(* IEC 61131-3 sources: SmartHomeNew/snapshots/2026-05-05, 45 files *)

(* ---- E_Lifetime_Device_Type.dut ---- *)
{attribute 'strict'}
TYPE E_Lifetime_Device_Type :
(
    LIFETIME_DEVICE_PUMP := 1,
    LIFETIME_DEVICE_FAN  := 2
) USINT;
END_TYPE

(* ---- E_Rule_Action_Type.dut ---- *)
{attribute 'strict'}
TYPE E_Rule_Action_Type :
(
    ACTION_NONE := 0,
    ACTION_SET_FLOOR_HEATING := 1,
    ACTION_SET_LIGHTING_BASE := 2,
    ACTION_SET_LIGHTING_ACCENT := 3,
    ACTION_SET_SOCKET := 4,
    ACTION_SET_VENTILATION := 5,
    ACTION_SET_BLINDS := 6,
    ACTION_ACTIVATE_SCENARIO := 7,
    ACTION_TOGGLE_LIGHTING := 8,
    ACTION_TOGGLE_SOCKET := 9
) USINT;
END_TYPE

(* ---- E_SCENARIO_SOURCE.dut ---- *)
TYPE E_SCENARIO_SOURCE :
(
    SRC_NONE := 0,
    SRC_OPERATOR := 1,
    SRC_GATEWAY := 2,
    SRC_RULE := 3,
    SRC_SAFETY := 4,
    SRC_POLICY := 5
);
END_TYPE

(* ---- E_System_Severity.dut ---- *)
TYPE E_System_Severity :
(
    SEV_NORMAL,
    SEV_WARNING,
    SEV_DEGRADED,
    SEV_CRITICAL
);
END_TYPE

(* ---- E_Trace_Source.dut ---- *)
{attribute 'strict'}
TYPE E_Trace_Source :
(
    SRC_MAIN := 0,
    SRC_IO := 1,
    SRC_DIAGNOSTICS := 2,
    SRC_HEATING := 3,
    SRC_SCENARIO := 4,
    SRC_USER := 5
) USINT;
END_TYPE

(* ---- GVL_SAFETY_SHUTDOWN.gvl ---- *)
TYPE E_Safety_Mode :
(
    NORMAL,
    FIRE,
    GAS,
    WATER_LEAK,
    GLOBAL_STOP,
    EVACUATION
);
END_TYPE

VAR_GLOBAL
    G_Safety_Mode : E_Safety_Mode := NORMAL;
    G_Safety_Active : BOOL := FALSE;
END_VAR

(* ---- GVL_CONFIG_CONTROL.gvl ---- *)
{attribute 'qualified_only'}
VAR_GLOBAL
    // Config change control. HMI/service writes here, never directly to active safety config.

    G_Apply_Request : BOOL := FALSE;
    G_Apply_Confirm : BOOL := FALSE;
    G_Rollback_Request : BOOL := FALSE;
    G_Rollback_Confirm : BOOL := FALSE;
    G_Reset_Default_Request : BOOL := FALSE;
    G_Reset_Default_Confirm : BOOL := FALSE;

    G_Config_Version : UDINT := 1;
    G_Last_Good_Version : UDINT := 1;
    G_Backup_Valid : BOOL := FALSE;
    G_Apply_Done : BOOL := FALSE;
    G_Rollback_Done : BOOL := FALSE;

    // STAGED INPUT CONFIG
    STG_Reputation_Learning_Rate : REAL := 0.05;
    STG_Reputation_Recovery_Decay : REAL := 0.01;
    STG_Min_Sensor_Confidence : REAL := 0.1;
    STG_Bad_Spike_Confidence : REAL := 0.3;
    STG_Default_Confidence : REAL := 1.0;

    // STAGED SCENARIO CONFIG
    STG_Night_Start_Hour : INT := 22;
    STG_Night_End_Hour : INT := 6;
    STG_VentBoost_Humidity_Threshold : REAL := 65.0;

    // STAGED RECOVERY CONFIG
    STG_Stabilization_Delay_MS : UDINT := 5000;

    // STAGED COMMAND POLICY CRITICAL PART
    STG_PLC_Inactive_Close_Gas : BOOL := TRUE;
    STG_PLC_Inactive_Stop_Boiler : BOOL := TRUE;
    STG_PLC_Inactive_Block_Heating : BOOL := TRUE;
    STG_PLC_Inactive_Stop_Vent : BOOL := TRUE;
    STG_PLC_Inactive_Block_Water : BOOL := TRUE;

    // BACKUP INPUT CONFIG
    BCK_Reputation_Learning_Rate : REAL := 0.05;
    BCK_Reputation_Recovery_Decay : REAL := 0.01;
    BCK_Min_Sensor_Confidence : REAL := 0.1;
    BCK_Bad_Spike_Confidence : REAL := 0.3;
    BCK_Default_Confidence : REAL := 1.0;

    // BACKUP SCENARIO CONFIG
    BCK_Night_Start_Hour : INT := 22;
    BCK_Night_End_Hour : INT := 6;
    BCK_VentBoost_Humidity_Threshold : REAL := 65.0;

    // BACKUP RECOVERY CONFIG
    BCK_Stabilization_Delay_MS : UDINT := 5000;

    // BACKUP COMMAND POLICY CRITICAL PART
    BCK_PLC_Inactive_Close_Gas : BOOL := TRUE;
    BCK_PLC_Inactive_Stop_Boiler : BOOL := TRUE;
    BCK_PLC_Inactive_Block_Heating : BOOL := TRUE;
    BCK_PLC_Inactive_Stop_Vent : BOOL := TRUE;
    BCK_PLC_Inactive_Block_Water : BOOL := TRUE;
END_VAR

(* ---- GVL_HEATING_OUTPUT.gvl ---- *)
VAR_GLOBAL
    // Heating output projection produced by PRG_Heating and consumed by PRG_IO_Write.
    // This removes the direct PRG_IO_Write -> GVL_STATE dependency for Heating physical outputs.

    DO_Zone_Valves : ARRAY[1..GVL_CONSTANTS.C_MAX_HEATING_CIRCUITS] OF BOOL;
    DO_Manifold_Pumps : ARRAY[1..GVL_CONSTANTS.C_MAX_MANIFOLDS] OF BOOL;
    AO_Manifold_Valves : ARRAY[1..GVL_CONSTANTS.C_MAX_MANIFOLDS] OF UINT;

    DO_DHW_Heating_Pump : BOOL := FALSE;
    DO_DHW_Circ_Pump : BOOL := FALSE;
    DO_Backup_Circulation_Pump : BOOL := FALSE;
    DO_Electric_Heater_Enable : BOOL := FALSE;
END_VAR

(* ---- GVL_HMI.gvl ---- *)
{attribute 'qualified_only'}
VAR_GLOBAL
    // Heating dashboard
    G_HMI_Heating_Confidence : REAL := 1.0;
    G_HMI_Heating_Confidence_Percent : INT := 100;
    G_HMI_Heating_Reason_Code : INT := 0;
    G_HMI_Heating_Status_Text : STRING(128) := 'OK';
    G_HMI_Heating_Status_Level : INT := 0; // 0=OK, 1=WARN, 2=ALARM

    // Heating predictive dashboard
    G_HMI_Heating_Predictive_Pressure_Drop : ARRAY[1..GVL_CONSTANTS.C_MAX_MANIFOLDS] OF BOOL;
    G_HMI_Heating_Predictive_Current_Rise : ARRAY[1..GVL_CONSTANTS.C_MAX_MANIFOLDS] OF BOOL;
END_VAR

(* ---- GVL_INTENT_BEHAVIOR.gvl ---- *)
VAR_GLOBAL
    // Behavior / Scenario Engine intent layer.
    // Scenario Engine writes here; Command Arbitration may consume it.

    I_Request_Night_Mode : BOOL := FALSE;
    I_Request_Away_Mode : BOOL := FALSE;
    I_Request_Comfort_Mode : BOOL := FALSE;
    I_Request_Energy_Save_Mode : BOOL := FALSE;
    I_Request_Preheat : BOOL := FALSE;
    I_Request_Ventilation_Boost : BOOL := FALSE;
    I_Request_Access_Secure_Mode : BOOL := FALSE;

    I_Target_Comfort_Temperature : REAL := 21.0;
    I_Behavior_Priority : INT := 0;

    // Candidate scenario scores for explainability / diagnostics
    I_Score_Comfort : INT := 0;
    I_Score_Night : INT := 0;
    I_Score_Energy_Save : INT := 0;
    I_Score_Preheat : INT := 0;
    I_Score_Vent_Boost : INT := 0;
    I_Score_Access_Secure : INT := 0;

    // Multi-objective weights, normalized 0.0..1.0 for HMI / downstream blending.
    I_Weight_Comfort : REAL := 0.0;
    I_Weight_Night : REAL := 0.0;
    I_Weight_Energy_Save : REAL := 0.0;
    I_Weight_Preheat : REAL := 0.0;
    I_Weight_Vent_Boost : REAL := 0.0;
    I_Weight_Access_Secure : REAL := 0.0;

    I_Best_VentBoost_Zone : INT := 0;

    I_Selected_Scenario_Code : E_System_Reason_Code := REASON_NONE;
    I_Selected_Scenario_Text : STRING(255) := 'No behavior scenario selected';

    I_Reason_Code : E_System_Reason_Code := REASON_NONE;
    I_Reason_Text : STRING(255) := 'No behavior scenario active';
    I_Last_Update_MS : UDINT := 0;
END_VAR

(* ---- GVL_INTENT_SAFETY.gvl ---- *)
VAR_GLOBAL
    // --- meta / traceability ---
    I_Source_Valid : BOOL := FALSE;
    I_Last_Update_Cycle : UDINT := 0;
    I_Last_Update_MS : UDINT := 0;

    // --- safety facts for arbitration ---
    I_Fire_Alarm_Active : BOOL := FALSE;
    I_Gas_Alarm_Active : BOOL := FALSE;
    I_Leak_Alarm_Active : BOOL := FALSE;
    I_CO_Warning_Active : BOOL := FALSE;
    I_System_Safe_Stop_Required : BOOL := FALSE;
    I_Freeze_Protection_Required : BOOL := FALSE;
    I_Evacuation_Mode_Active : BOOL := FALSE;

    // --- gas / boiler / ventilation constraints ---
    I_Gas_Close_Required : BOOL := FALSE;
    I_Boiler_Stop_Required : BOOL := FALSE;
    I_Vent_Stop_Required : BOOL := FALSE;
    I_Vent_Force_PV3_Boost : BOOL := FALSE;
    I_Vent_Force_Supply_100 : BOOL := FALSE;
    I_Vent_Force_Supply_80 : BOOL := FALSE;
    I_Vent_Force_Exhaust_100 : BOOL := FALSE;

    // --- water constraints ---
    I_Water_Main_Close_Required : BOOL := FALSE;
    I_Water_Zone_Close_Required : ARRAY[1..32] OF BOOL;
    I_Water_Selective_Recovery_Allowed : BOOL := FALSE;
    I_Water_Recovery_Target_Zone : INT := 0;

    // --- lock / evacuation constraints ---
    I_Lock_1_Force_Open : BOOL := FALSE;
    I_Lock_1_Force_Close_Block : BOOL := FALSE;
    I_Lock_2_Force_Open : BOOL := FALSE;
    I_Lock_2_Force_Close_Block : BOOL := FALSE;
    // --- operator / test constraints ---
    I_Test_Timeout_Gas_Close : BOOL := FALSE;
    I_Test_Timeout_Water_Close : BOOL := FALSE;
END_VAR

(* ---- GVL_SIMULATION.gvl ---- *)
{attribute 'qualified_only'}
VAR_GLOBAL
    G_Simulation_Enable : BOOL := FALSE;

    // Scenario control
    G_Test_Scenario_ID : INT := 0; // 0=manual flags, 1=safety gas, 2=leak+low pressure, 3=sensor+predictive, 4=dual PLC, 5=full stress
    G_Test_Start : BOOL := FALSE;
    G_Test_Stop : BOOL := FALSE;
    G_Test_Scenario_Active : BOOL := FALSE;
    G_Test_Started_MS : UDINT := 0;
    G_Test_Duration_MS : UDINT := 30000;
    G_Test_Expected_Result_Code : INT := 0; // 0=none, 1=safety, 2=heating degraded, 3=role conflict, 4=full stress

    // Sensor fault injection requests
    G_Inject_Heating_Sensor_Fault : BOOL := FALSE;
    G_Inject_IO_Fault : BOOL := FALSE;
    G_Inject_Low_Pressure : BOOL := FALSE;
    G_Inject_Predictive_Pump_Fault : BOOL := FALSE;

    // Safety fault injection requests
    G_Inject_Gas_Alarm : BOOL := FALSE;
    G_Inject_Leak_Alarm : BOOL := FALSE;
    G_Inject_Smoke_Alarm : BOOL := FALSE;

    // PLC / role fault injection request
    G_Inject_Dual_PLC_Active : BOOL := FALSE;

    // Isolated effective simulation outputs. Production state is not overwritten by PRG_System_Simulation.
    G_Sim_Heating_Sensor_Fault : BOOL := FALSE;
    G_Sim_IO_Fault : BOOL := FALSE;
    G_Sim_Low_Pressure : BOOL := FALSE;
    G_Sim_Predictive_Pump_Fault : BOOL := FALSE;
    G_Sim_Gas_Alarm : BOOL := FALSE;
    G_Sim_Leak_Alarm : BOOL := FALSE;
    G_Sim_Smoke_Alarm : BOOL := FALSE;
    G_Sim_Dual_PLC_Active : BOOL := FALSE;

    // Test status
    G_Test_Running : BOOL := FALSE;
    G_Test_Result_OK : BOOL := FALSE;
    G_Test_Last_Result_Text : STRING(128) := 'No test executed';
END_VAR

(* ---- GVL_SYSTEM_SIZE_CONFIG.gvl ---- *)
{attribute 'qualified_only'}
VAR_GLOBAL
    // Runtime active counts. Arrays remain allocated by GVL_CONSTANTS.C_MAX_*.
    // These values define how many channels/zones are actively processed.

    G_Active_Heating_Circuits : INT := GVL_CONSTANTS.C_MAX_HEATING_CIRCUITS;
    G_Active_Water_Zones : INT := GVL_CONSTANTS.C_MAX_WATER_ZONES;
    G_Active_Light_Zones : INT := GVL_CONSTANTS.C_MAX_LIGHT_ZONES;
    G_Active_Blinds : INT := GVL_CONSTANTS.C_MAX_BLINDS;
    G_Active_Sockets : INT := GVL_CONSTANTS.C_MAX_SOCKETS;
END_VAR

(* ---- FB_Boiler_OpenTherm_Interface.st ---- *)
FUNCTION_BLOCK FB_Boiler_OpenTherm_Interface
VAR_INPUT
    VI_Enable : ARRAY[1..GVL_CONSTANTS.C_MAX_BOILERS] OF BOOL;
    VI_Setpoint : ARRAY[1..GVL_CONSTANTS.C_MAX_BOILERS] OF REAL;

    VI_OT_Online : ARRAY[1..GVL_CONSTANTS.C_MAX_BOILERS] OF BOOL;
    VI_OT_Error : ARRAY[1..GVL_CONSTANTS.C_MAX_BOILERS] OF BOOL;
END_VAR

VAR_OUTPUT
    VO_OT_Enable : ARRAY[1..GVL_CONSTANTS.C_MAX_BOILERS] OF BOOL;
    VO_OT_Setpoint : ARRAY[1..GVL_CONSTANTS.C_MAX_BOILERS] OF REAL;
    VO_OT_Command_Valid : ARRAY[1..GVL_CONSTANTS.C_MAX_BOILERS] OF BOOL;
END_VAR

VAR
    L_i : INT;
END_VAR

FOR L_i := 1 TO GVL_CONSTANTS.C_MAX_BOILERS DO
    VO_OT_Enable[L_i] := FALSE;
    VO_OT_Setpoint[L_i] := 0.0;
    VO_OT_Command_Valid[L_i] := FALSE;

    IF VI_Enable[L_i] AND VI_OT_Online[L_i] AND NOT VI_OT_Error[L_i] THEN
        VO_OT_Enable[L_i] := TRUE;
        VO_OT_Setpoint[L_i] := LIMIT(20.0, VI_Setpoint[L_i], 80.0);
        VO_OT_Command_Valid[L_i] := TRUE;
    END_IF;
END_FOR;
END_FUNCTION_BLOCK

(* ---- FB_Calibration_Manager.st ---- *)
FUNCTION_BLOCK FB_Calibration_Manager
VAR_INPUT
    VI_Raw_Value : REAL;
    VI_Type : BYTE; // 1-Temp, 2-Pressure, 3-Gas
    VI_Calib_Record : ST_Sensor_Calibration_Record;
    VI_System_Time_MS : UDINT;
    VI_Start_Verification : BOOL;
END_VAR
VAR_OUTPUT
    VO_Calibrated_Value : REAL;
    VO_Verification_Active : BOOL;
    VO_Verification_Failed : BOOL;
    VO_Deviation_Percent : REAL;
END_VAR
VAR
    L_Verification_Timer : FB_System_Timer;
    L_Initial_Value : REAL;
END_VAR

// 1. Расчет калиброванного значения
CASE VI_Type OF
    1: VO_Calibrated_Value := VI_Raw_Value + VI_Calib_Record.offset;
    2, 3: VO_Calibrated_Value := (VI_Raw_Value * VI_Calib_Record.multiplier) + VI_Calib_Record.offset;
END_CASE;

// 2. Верификация через 1 час (ТЗ 9.5)
IF VI_Start_Verification AND NOT VO_Verification_Active THEN
    VO_Verification_Active := TRUE;
    L_Initial_Value := VO_Calibrated_Value;
END_IF;

L_Verification_Timer(IN := VO_Verification_Active, PT := T#1h, VI_System_Time_MS := VI_System_Time_MS);

IF L_Verification_Timer.Q THEN
    VO_Verification_Active := FALSE;

    // ТЗ 9.5: Отклонение ≤2.0% (норма) / >5.0% (ошибка)
    IF L_Initial_Value <> 0 THEN
        VO_Deviation_Percent := ABS(VO_Calibrated_Value - L_Initial_Value) / L_Initial_Value * 100.0;
    ELSE
        VO_Deviation_Percent := 0.0;
    END_IF;

    VO_Verification_Failed := (VO_Deviation_Percent > 5.0);
END_IF;
END_FUNCTION_BLOCK

(* ---- FB_Fault_Logger.st ---- *)
FUNCTION_BLOCK FB_Fault_Logger
VAR_INPUT
    VI_Severity  : E_System_Severity;
    VI_RootCause : E_System_Root_Cause;
    VI_Time_MS   : UDINT;
END_VAR

VAR_OUTPUT
    VO_Last_Event_Text : STRING(200);
    VO_Event_Count     : UINT;
    VO_Last_Index      : UINT;

    VO_Event_Time_MS   : ARRAY[1..16] OF UDINT;
    VO_Event_Severity  : ARRAY[1..16] OF E_System_Severity;
    VO_Event_RootCause : ARRAY[1..16] OF E_System_Root_Cause;
    VO_Event_Text      : ARRAY[1..16] OF STRING(200);
END_VAR

VAR
    L_Last_Severity  : E_System_Severity;
    L_Last_RootCause : E_System_Root_Cause;
    L_Write_Index    : UINT := 0;
    L_Event_Text     : STRING(200);
END_VAR

L_Event_Text := '';

IF (VI_Severity <> L_Last_Severity) OR (VI_RootCause <> L_Last_RootCause) THEN
    CASE VI_RootCause OF
        E_System_Root_Cause.ROOT_FIRE:
            L_Event_Text := 'EVENT: FIRE DETECTED';
        E_System_Root_Cause.ROOT_GAS_LEAK:
            L_Event_Text := 'EVENT: GAS LEAK';
        E_System_Root_Cause.ROOT_CO_CRITICAL:
            L_Event_Text := 'EVENT: CO CRITICAL';
        E_System_Root_Cause.ROOT_CO_WARNING:
            L_Event_Text := 'EVENT: CO WARNING';
        E_System_Root_Cause.ROOT_WATER_LEAK:
            L_Event_Text := 'EVENT: WATER LEAK';
        E_System_Root_Cause.ROOT_SENSOR_FAULT:
            L_Event_Text := 'EVENT: SENSOR FAULT';
        E_System_Root_Cause.ROOT_IO_OFFLINE:
            L_Event_Text := 'EVENT: IO OFFLINE';
        E_System_Root_Cause.ROOT_COMM_FAULT:
            L_Event_Text := 'EVENT: COMM FAULT';
        E_System_Root_Cause.ROOT_WATCHDOG_FAULT:
            L_Event_Text := 'EVENT: WATCHDOG FAULT';
        E_System_Root_Cause.ROOT_SUBSYSTEM_FAULT:
            L_Event_Text := 'EVENT: SUBSYSTEM FAULT';
        ELSE
            L_Event_Text := 'EVENT: SYSTEM STATE CHANGE';
    END_CASE;

    L_Write_Index := L_Write_Index + 1;
    IF L_Write_Index > 16 THEN
        L_Write_Index := 1;
    END_IF;

    VO_Event_Time_MS[L_Write_Index] := VI_Time_MS;
    VO_Event_Severity[L_Write_Index] := VI_Severity;
    VO_Event_RootCause[L_Write_Index] := VI_RootCause;
    VO_Event_Text[L_Write_Index] := L_Event_Text;

    VO_Last_Index := L_Write_Index;
    VO_Last_Event_Text := L_Event_Text;

    IF VO_Event_Count < 16 THEN
        VO_Event_Count := VO_Event_Count + 1;
    END_IF;
END_IF;

L_Last_Severity := VI_Severity;
L_Last_RootCause := VI_RootCause;
// >>> BULK_SYNC_ANCHOR: FB_Fault_Logger <<<
END_FUNCTION_BLOCK

(* ---- FB_FloorHeating_Overheat_Protection.st ---- *)
FUNCTION_BLOCK FB_FloorHeating_Overheat_Protection
VAR_INPUT
    VI_Threshold : REAL := 45.0;
END_VAR
VAR_IN_OUT
    VI_Temps : ARRAY[1..GVL_CONSTANTS.C_MAX_HEATING_CIRCUITS] OF REAL;
END_VAR
VAR_OUTPUT
    VO_Overheat_Detected : BOOL;
    VO_Locked_Circuits : ARRAY[1..GVL_CONSTANTS.C_MAX_HEATING_CIRCUITS] OF BOOL;
END_VAR
VAR
    L_i : INT;
END_VAR

VO_Overheat_Detected := FALSE;
FOR L_i := 1 TO GVL_CONSTANTS.C_MAX_HEATING_CIRCUITS DO
    IF VI_Temps[L_i] > VI_Threshold THEN
        VO_Overheat_Detected := TRUE;
        VO_Locked_Circuits[L_i] := TRUE;
    END_IF;
END_FOR;
END_FUNCTION_BLOCK

(* ---- FB_Gateway_Interface.st ---- *)
FUNCTION_BLOCK FB_Gateway_Interface
VAR_INPUT
    VI_System_Time_MS           : UDINT;
    VI_Local_PLC_Role           : E_PLC_ROLE;
    VI_Incoming_Command         : ST_Gateway_Command;
    VI_Command_Received         : BOOL;
    VI_Outdoor_Temp             : REAL;
    VI_Security_Armed           : BOOL;
    VI_Flood_Alarm_Active       : BOOL;
    VI_Gas_Alarm_Active         : BOOL;
    VI_Fire_Alarm_Active        : BOOL;
    VI_Methane_Concentration    : REAL;
    VI_Active_Scenario          : E_SCENARIO_TYPE;
    VI_Send_2FA_Req             : BOOL;
    VI_2FA_Code                 : STRING(6);
END_VAR

VAR_IN_OUT
    VI_FloorHeating_Temps       : ARRAY[1..GVL_CONSTANTS.C_MAX_HEATING_CIRCUITS] OF REAL;
    VI_Room_Temps               : ARRAY[1..GVL_CONSTANTS.C_MAX_ZONES] OF REAL;
    VI_Zone_Valve_States        : ARRAY[1..GVL_CONSTANTS.C_MAX_HEATING_CIRCUITS] OF BOOL;
    VI_Manifold_Pressures       : ARRAY[1..GVL_CONSTANTS.C_MAX_MANIFOLDS] OF REAL;
    VI_Manifold_Pump_States     : ARRAY[1..GVL_CONSTANTS.C_MAX_MANIFOLDS] OF BOOL;
    VI_Lighting_Base_Levels     : ARRAY[1..GVL_CONSTANTS.C_MAX_LIGHT_ZONES] OF BYTE;
    VI_Socket_States            : ARRAY[1..GVL_CONSTANTS.C_MAX_SOCKETS] OF BOOL;
    VI_Blinds_Positions         : ARRAY[1..GVL_CONSTANTS.C_MAX_BLINDS] OF BYTE;
    VI_Allowed_IPs              : ARRAY[1..GVL_CONSTANTS.C_MAX_ALLOWED_IPS] OF STRING(15);
END_VAR

VAR_OUTPUT
    VO_Modbus_Registers         : ARRAY[0..GVL_CONSTANTS.C_MAX_MODBUS_REGISTERS-1] OF WORD;
    VO_Lighting_Override        : ARRAY[1..GVL_CONSTANTS.C_MAX_LIGHT_ZONES] OF BYTE;
    VO_Blinds_Override          : ARRAY[1..GVL_CONSTANTS.C_MAX_BLINDS] OF BYTE;
    VO_Socket_Override          : ARRAY[1..GVL_CONSTANTS.C_MAX_SOCKETS] OF BOOL;
    VO_Arm_Req                  : BOOL;
    VO_Disarm_Req               : BOOL;
    VO_PIN_Code                 : STRING(4);
    VO_RFID_Tag                 : STRING(20);
    VO_2FA_Code_In              : STRING(6);
    VO_Data_Ready               : BOOL;
    VO_HMI_Status_Message       : STRING(200);
    VO_Telegram_Msg             : STRING(200);
    VO_Send_Telegram            : BOOL;
    VO_Set_Scenario_Req         : BOOL;
    VO_Target_Scenario          : E_SCENARIO_TYPE;
    VO_Set_Temp_Req             : BOOL;
    VO_Target_Zone              : INT;
    VO_Target_Temp              : REAL;
    VO_Set_Vent_Req             : BOOL;
    VO_Target_Vent_Speed        : BYTE;
    VO_Reset_Errors_Req         : BOOL;
    VO_Set_Config_Req           : BOOL;
    VO_Sync_Time_Req            : BOOL;
    VO_New_Time_MS              : UDINT;
END_VAR

VAR
    L_last_update_time          : UDINT;
    L_i                         : INT;
    L_j                         : INT;
    L_idx                       : INT;
    L_tmp_word                  : WORD;
    L_Code_UDINT                : UDINT;
    L_Prev_Fire                 : BOOL;
    L_Prev_Gas                  : BOOL;
    L_Prev_Flood                : BOOL;
    L_Prev_Security             : BOOL;
    L_Deduplicator              : FB_Command_Deduplication;
    L_CRC_Calc                  : FB_CRC32_Calculator;
    L_Calculated_CRC            : DWORD;
    L_IP_Allowed                : BOOL;
    L_Process_Command           : ST_Gateway_Command;
    L_Has_Command_To_Process    : BOOL;
END_VAR

VAR RETAIN
    L_Command_Buffer            : ARRAY[1..GVL_CONSTANTS.C_MAX_GATEWAY_COMMANDS] OF ST_Gateway_Command;
    L_Buffer_Head               : INT := 1;
    L_Buffer_Tail               : INT := 1;
    L_Buffer_Count              : INT := 0;
END_VAR

VO_Send_Telegram := FALSE;
IF VI_Fire_Alarm_Active AND NOT L_Prev_Fire THEN
    VO_Telegram_Msg := 'ВНИМАНИЕ! ПОЖАРНАЯ ТРЕВОГА!';
    VO_Send_Telegram := TRUE;
END_IF;
IF VI_Gas_Alarm_Active AND NOT L_Prev_Gas THEN
    VO_Telegram_Msg := 'ВНИМАНИЕ! УТЕЧКА ГАЗА!';
    VO_Send_Telegram := TRUE;
END_IF;
IF VI_Flood_Alarm_Active AND NOT L_Prev_Flood THEN
    VO_Telegram_Msg := 'ВНИМАНИЕ! ПРОТЕЧКА ВОДЫ!';
    VO_Send_Telegram := TRUE;
END_IF;
IF VI_Security_Armed AND NOT L_Prev_Security THEN
    VO_Telegram_Msg := 'ОХРАНА ВКЛЮЧЕНА';
    VO_Send_Telegram := TRUE;
ELSIF NOT VI_Security_Armed AND L_Prev_Security THEN
    VO_Telegram_Msg := 'ОХРАНА ОТКЛЮЧЕНА';
    VO_Send_Telegram := TRUE;
END_IF;

L_Prev_Fire := VI_Fire_Alarm_Active;
L_Prev_Gas := VI_Gas_Alarm_Active;
L_Prev_Flood := VI_Flood_Alarm_Active;
L_Prev_Security := VI_Security_Armed;

IF (VI_System_Time_MS - L_last_update_time) >= GVL_CONSTANTS.C_MS_IN_SECOND THEN
    L_last_update_time := VI_System_Time_MS;
    L_tmp_word := 0;
    IF VI_Local_PLC_Role = E_PLC_ROLE.ROLE_ACTIVE THEN L_tmp_word := L_tmp_word OR 1; END_IF;
    IF VI_Security_Armed THEN L_tmp_word := L_tmp_word OR 2; END_IF;
    IF VI_Flood_Alarm_Active THEN L_tmp_word := L_tmp_word OR 4; END_IF;
    IF VI_Gas_Alarm_Active THEN L_tmp_word := L_tmp_word OR 8; END_IF;
    IF VI_Fire_Alarm_Active THEN L_tmp_word := L_tmp_word OR 16; END_IF;
    VO_Modbus_Registers[0] := L_tmp_word;

    FOR L_i := 1 TO GVL_CONSTANTS.C_MAX_HEATING_CIRCUITS DO
        VO_Modbus_Registers[L_i] := TO_WORD(TO_INT(VI_FloorHeating_Temps[L_i] * REAL#10.0));
    END_FOR;

    FOR L_i := 1 TO GVL_CONSTANTS.C_MAX_ZONES DO
        VO_Modbus_Registers[16 + L_i] := TO_WORD(TO_INT(VI_Room_Temps[L_i] * REAL#10.0));
    END_FOR;

    L_tmp_word := 0;
    FOR L_i := 1 TO GVL_CONSTANTS.C_MAX_HEATING_CIRCUITS DO
        IF VI_Zone_Valve_States[L_i] THEN
            L_tmp_word := L_tmp_word OR SHL(TO_WORD(1), L_i - 1);
        END_IF;
    END_FOR;
    VO_Modbus_Registers[33] := L_tmp_word;

    FOR L_i := 1 TO GVL_CONSTANTS.C_MAX_MANIFOLDS DO
        VO_Modbus_Registers[33 + L_i] := TO_WORD(TO_INT(VI_Manifold_Pressures[L_i] * REAL#100.0));
    END_FOR;

    FOR L_i := 1 TO GVL_CONSTANTS.C_MAX_LIGHT_ZONES DO
        VO_Modbus_Registers[39 + L_i] := TO_WORD(VI_Lighting_Base_Levels[L_i]);
    END_FOR;

    FOR L_i := 1 TO GVL_CONSTANTS.C_MAX_BLINDS DO
        VO_Modbus_Registers[71 + L_i] := TO_WORD(VI_Blinds_Positions[L_i]);
    END_FOR;

    FOR L_i := 0 TO (GVL_CONSTANTS.C_MAX_SOCKETS - 1) / 16 DO
        L_tmp_word := 0;
        FOR L_j := 1 TO 16 DO
            L_idx := (L_i * 16) + L_j;
            IF L_idx <= GVL_CONSTANTS.C_MAX_SOCKETS THEN
                IF VI_Socket_States[L_idx] THEN
                    L_tmp_word := L_tmp_word OR SHL(TO_WORD(1), L_j - 1);
                END_IF;
            END_IF;
        END_FOR;
        VO_Modbus_Registers[92 + L_i] := L_tmp_word;
    END_FOR;

    VO_Modbus_Registers[100] := SEL(VI_Send_2FA_Req, 0, 1);
    IF VI_Send_2FA_Req THEN
        L_Code_UDINT := STRING_TO_UDINT(VI_2FA_Code);
        VO_Modbus_Registers[101] := TO_WORD(L_Code_UDINT AND 16#FFFF);
        VO_Modbus_Registers[102] := TO_WORD(SHR(L_Code_UDINT, 16));
    ELSE
        VO_Modbus_Registers[101] := 0;
        VO_Modbus_Registers[102] := 0;
    END_IF;

    VO_Data_Ready := TRUE;
END_IF;

VO_Arm_Req := FALSE;
VO_Disarm_Req := FALSE;
VO_Set_Scenario_Req := FALSE;
VO_Set_Temp_Req := FALSE;
VO_Set_Vent_Req := FALSE;
VO_Reset_Errors_Req := FALSE;
VO_Set_Config_Req := FALSE;
VO_Sync_Time_Req := FALSE;
L_Has_Command_To_Process := FALSE;

IF VI_Command_Received THEN
    IF VI_Local_PLC_Role = E_PLC_ROLE.ROLE_ACTIVE THEN
        L_Process_Command := VI_Incoming_Command;
        L_Has_Command_To_Process := TRUE;
    ELSE
        IF L_Buffer_Count < GVL_CONSTANTS.C_MAX_GATEWAY_COMMANDS THEN
            L_Command_Buffer[L_Buffer_Head] := VI_Incoming_Command;
            L_Buffer_Head := L_Buffer_Head + 1;
            IF L_Buffer_Head > GVL_CONSTANTS.C_MAX_GATEWAY_COMMANDS THEN L_Buffer_Head := 1; END_IF;
            L_Buffer_Count := L_Buffer_Count + 1;
        END_IF;
    END_IF;
END_IF;

IF NOT L_Has_Command_To_Process AND (VI_Local_PLC_Role = E_PLC_ROLE.ROLE_ACTIVE) AND (L_Buffer_Count > 0) THEN
    L_Process_Command := L_Command_Buffer[L_Buffer_Tail];
    L_Buffer_Tail := L_Buffer_Tail + 1;
    IF L_Buffer_Tail > GVL_CONSTANTS.C_MAX_GATEWAY_COMMANDS THEN L_Buffer_Tail := 1; END_IF;
    L_Buffer_Count := L_Buffer_Count - 1;
    L_Has_Command_To_Process := TRUE;
END_IF;

IF L_Has_Command_To_Process THEN
    L_IP_Allowed := FALSE;
    IF L_Process_Command.source_ip = '' THEN
        L_IP_Allowed := TRUE;
    ELSE
        FOR L_i := 1 TO GVL_CONSTANTS.C_MAX_ALLOWED_IPS DO
            IF VI_Allowed_IPs[L_i] = L_Process_Command.source_ip THEN
                L_IP_Allowed := TRUE;
                EXIT;
            END_IF;
        END_FOR;
    END_IF;

    IF NOT L_IP_Allowed THEN
        VO_HMI_Status_Message := 'Gateway: Ошибка безопасности (Неизвестный IP)';
        RETURN;
    END_IF;

    L_CRC_Calc();
    L_Calculated_CRC := L_CRC_Calc.VO_CRC;

    IF L_Calculated_CRC = L_Process_Command.crc32 THEN
        L_Deduplicator(VI_Command_ID := L_Process_Command.command_id, VI_Command_Type := L_Process_Command.command_type, VI_Command_Value := L_Process_Command.target_value, VI_System_Time_MS := VI_System_Time_MS);

        IF L_Deduplicator.VO_Is_New_Command THEN
            CASE L_Process_Command.command_type OF
                E_Gateway_Command_Type.CMD_SET_SCENARIO:
                    VO_Set_Scenario_Req := TRUE;
                    VO_Target_Scenario := L_Process_Command.target_scenario;
                    VO_HMI_Status_Message := 'Gateway: Сценарий изменен';
                E_Gateway_Command_Type.CMD_SET_LIGHT:
                    IF (L_Process_Command.target_zone >= 1) AND (L_Process_Command.target_zone <= GVL_CONSTANTS.C_MAX_LIGHT_ZONES) THEN
                        VO_Lighting_Override[L_Process_Command.target_zone] := TO_BYTE(L_Process_Command.target_value);
                        VO_HMI_Status_Message := 'Gateway: Команда освещения принята';
                    END_IF;
                E_Gateway_Command_Type.CMD_SET_BLINDS:
                    IF (L_Process_Command.target_zone >= 1) AND (L_Process_Command.target_zone <= GVL_CONSTANTS.C_MAX_BLINDS) THEN
                        VO_Blinds_Override[L_Process_Command.target_zone] := TO_BYTE(L_Process_Command.target_value);
                        VO_HMI_Status_Message := 'Gateway: Команда штор принята';
                    END_IF;
                E_Gateway_Command_Type.CMD_SET_SOCKET:
                    IF (L_Process_Command.target_zone >= 1) AND (L_Process_Command.target_zone <= GVL_CONSTANTS.C_MAX_SOCKETS) THEN
                        VO_Socket_Override[L_Process_Command.target_zone] := L_Process_Command.target_on_off;
                        VO_HMI_Status_Message := 'Gateway: Команда розетки принята';
                    END_IF;
                E_Gateway_Command_Type.CMD_SET_SECURITY:
                    IF L_Process_Command.target_armed THEN VO_Arm_Req := TRUE; ELSE VO_Disarm_Req := TRUE; END_IF;
                    VO_PIN_Code := L_Process_Command.target_pin;
                    VO_2FA_Code_In := L_Process_Command.target_2fa_code;
                    VO_HMI_Status_Message := 'Gateway: Запрос охраны принят';
                E_Gateway_Command_Type.CMD_SET_TEMP:
                    IF (L_Process_Command.target_zone >= 1) AND (L_Process_Command.target_zone <= GVL_CONSTANTS.C_MAX_HEATING_CIRCUITS) THEN
                        VO_Set_Temp_Req := TRUE;
                        VO_Target_Zone := L_Process_Command.target_zone;
                        VO_Target_Temp := L_Process_Command.target_value;
                        VO_HMI_Status_Message := 'Gateway: Уставка температуры изменена';
                    END_IF;
                E_Gateway_Command_Type.CMD_SET_VENT:
                    VO_Set_Vent_Req := TRUE;
                    VO_Target_Vent_Speed := TO_BYTE(L_Process_Command.target_value);
                    VO_HMI_Status_Message := 'Gateway: Уставка вентиляции изменена';
                E_Gateway_Command_Type.CMD_TELEGRAM_MSG:
                    VO_Telegram_Msg := L_Process_Command.telegram_msg;
                    VO_Send_Telegram := TRUE;
                    VO_HMI_Status_Message := 'Gateway: Сообщение Telegram отправлено';
                E_Gateway_Command_Type.CMD_SYNC_TIME:
                    VO_Sync_Time_Req := TRUE;
                    VO_New_Time_MS := REAL_TO_UDINT(L_Process_Command.target_value);
                    VO_HMI_Status_Message := 'Gateway: Время синхронизировано';
                E_Gateway_Command_Type.CMD_RESET_ERRORS:
                    VO_Reset_Errors_Req := TRUE;
                    VO_HMI_Status_Message := 'Gateway: Запрос на сброс ошибок принят';
                E_Gateway_Command_Type.CMD_SET_CONFIG:
                    VO_Set_Config_Req := TRUE;
                    VO_HMI_Status_Message := 'Gateway: Запрос на применение конфигурации принят';
            END_CASE;
        END_IF;
    ELSE
        VO_HMI_Status_Message := 'Gateway: Ошибка CRC команды';
    END_IF;
END_IF;

// >>> BULK_SYNC_ANCHOR: FB_Gateway_Interface <<<
END_FUNCTION_BLOCK

(* ---- FB_Heating_Boiler_Control.st ---- *)
// ==============================================================================
// Heating boiler control helper
// ==============================================================================
FUNCTION_BLOCK FB_Heating_Boiler_Control
VAR_INPUT
    VI_System_Time_MS : UDINT;
    VI_IsActivePLC : BOOL;
    VI_DHW_Heating_Demand : BOOL;
    VI_DHW_Target_Temp : REAL;
    VI_Target_Supply_Temp : REAL;
    VI_Freeze_Mode_Active : BOOL;
    VI_Policy_Degraded : BOOL;
    VI_Manifold_Pumps : ARRAY[1..GVL_CONSTANTS.C_MAX_MANIFOLDS] OF BOOL;
    VI_Manifold_Valves : ARRAY[1..GVL_CONSTANTS.C_MAX_MANIFOLDS] OF REAL;
    VI_Boiler_Flame_Status : ARRAY[1..GVL_CONSTANTS.C_MAX_BOILERS] OF BOOL;
    VI_Boiler_Error_Status : ARRAY[1..GVL_CONSTANTS.C_MAX_BOILERS] OF BOOL;
    VI_Boiler_OT_Online : ARRAY[1..GVL_CONSTANTS.C_MAX_BOILERS] OF BOOL;
END_VAR
VAR_IN_OUT
    VI_Boiler_Modulation : ARRAY[1..GVL_CONSTANTS.C_MAX_BOILERS] OF REAL;
END_VAR
VAR_OUTPUT
    VO_Boiler_OT_Enable : ARRAY[1..GVL_CONSTANTS.C_MAX_BOILERS] OF BOOL;
    VO_Boiler_OT_Setpoint : ARRAY[1..GVL_CONSTANTS.C_MAX_BOILERS] OF REAL;
    VO_Boiler_Status : ARRAY[1..GVL_CONSTANTS.C_MAX_BOILERS] OF ST_Boiler_Status;
    VO_Any_Subsystem_Degraded : BOOL;
    VO_Lead_Boiler : BYTE;
    VO_Demand_Power : REAL;
END_VAR
VAR
    L_i : INT;
    L_Delta_MS : UDINT;
    L_Last_Scan_Time : UDINT;
    L_Scan_Time_Init : BOOL := FALSE;
    L_Boiler_Request_Enable : ARRAY[1..GVL_CONSTANTS.C_MAX_BOILERS] OF BOOL;
    L_Boiler_Request_Setpoint : ARRAY[1..GVL_CONSTANTS.C_MAX_BOILERS] OF REAL;
    L_Boiler_OT_Command_Valid : ARRAY[1..GVL_CONSTANTS.C_MAX_BOILERS] OF BOOL;
    L_Boiler_Life : ARRAY[1..GVL_CONSTANTS.C_MAX_BOILERS] OF FB_Lifetime_Predictor;
    fbBoilerCascade : FB_Boiler_Cascade_Manager;
    fbBoilerOpenTherm : FB_Boiler_OpenTherm_Interface;
END_VAR

VO_Any_Subsystem_Degraded := FALSE;
VO_Demand_Power := 0.0;

FOR L_i := 1 TO GVL_CONSTANTS.C_MAX_MANIFOLDS DO
    IF VI_Manifold_Pumps[L_i] THEN
        VO_Demand_Power := VO_Demand_Power + VI_Manifold_Valves[L_i];
    END_IF;
END_FOR;

IF VI_Freeze_Mode_Active AND VO_Demand_Power < 20.0 THEN
    VO_Demand_Power := 20.0;
END_IF;

IF VI_Policy_Degraded THEN
    IF VO_Demand_Power > 60.0 THEN
        VO_Demand_Power := 60.0;
    END_IF;
END_IF;

fbBoilerCascade(
    VI_Enable := VI_IsActivePLC AND ((VO_Demand_Power > GVL_CONSTANTS.C_BOILER_CASCADE_MIN_DEMAND) OR VI_Freeze_Mode_Active),
    VI_System_Time_MS := VI_System_Time_MS,
    VI_Boiler_Stop := FALSE,
    VI_DHW_Heating_Demand := VI_DHW_Heating_Demand,
    VI_DHW_Target_Temp := VI_DHW_Target_Temp,
    VI_Target_Supply_Temp := VI_Target_Supply_Temp,
    VI_Demand_Power := VO_Demand_Power,
    VI_Boiler_Flame_Status := VI_Boiler_Flame_Status,
    VI_Boiler_Error_Status := VI_Boiler_Error_Status,
    VI_Boiler_OT_Online := VI_Boiler_OT_Online,
    VI_Boiler_Modulation := VI_Boiler_Modulation,
    VO_Boiler_Enable => L_Boiler_Request_Enable,
    VO_Boiler_Setpoint => L_Boiler_Request_Setpoint,
    VO_Lead_Boiler => VO_Lead_Boiler
);

// === SAFETY CLAMP (35–55°C) ===
FOR L_i := 1 TO GVL_CONSTANTS.C_MAX_BOILERS DO
    IF L_Boiler_Request_Enable[L_i] THEN
        L_Boiler_Request_Setpoint[L_i] := LIMIT(
            GVL_CONSTANTS.C_BOILER_SETPOINT_MIN,
            L_Boiler_Request_Setpoint[L_i],
            GVL_CONSTANTS.C_BOILER_SETPOINT_MAX
        );
    END_IF;
END_FOR;

FOR L_i := 1 TO GVL_CONSTANTS.C_MAX_BOILERS DO
    IF NOT VI_Boiler_OT_Online[L_i] OR VI_Boiler_Error_Status[L_i] THEN
        L_Boiler_Request_Enable[L_i] := FALSE;
        L_Boiler_Request_Setpoint[L_i] := 0.0;
    END_IF;
END_FOR;

fbBoilerOpenTherm(
    VI_Enable := L_Boiler_Request_Enable,
    VI_Setpoint := L_Boiler_Request_Setpoint,
    VI_OT_Online := VI_Boiler_OT_Online,
    VI_OT_Error := VI_Boiler_Error_Status,
    VO_OT_Enable => VO_Boiler_OT_Enable,
    VO_OT_Setpoint => VO_Boiler_OT_Setpoint,
    VO_OT_Command_Valid => L_Boiler_OT_Command_Valid
);

// (остальной код без изменений)

END_FUNCTION_BLOCK

(* ---- FB_Heating_Decision_Context.st ---- *)
FUNCTION_BLOCK FB_Heating_Decision_Context
VAR_INPUT
    VI_Manifold_Pump_In_Service : ARRAY[1..GVL_CONSTANTS.C_MAX_MANIFOLDS] OF BOOL;
    VI_Manifold_Pressure_Fault : ARRAY[1..GVL_CONSTANTS.C_MAX_MANIFOLDS] OF BOOL;
    VI_Manifold_Current_Fault : ARRAY[1..GVL_CONSTANTS.C_MAX_MANIFOLDS] OF BOOL;
    VI_Manifold_Thermal_Weight : ARRAY[1..GVL_CONSTANTS.C_MAX_MANIFOLDS] OF REAL;
    VI_Manifold_Priority : ARRAY[1..GVL_CONSTANTS.C_MAX_MANIFOLDS] OF INT;
    VI_Max_Thermal_Budget : REAL;
END_VAR
VAR_OUTPUT
    VO_Manifold_Allowed : ARRAY[1..GVL_CONSTANTS.C_MAX_MANIFOLDS] OF BOOL;
    VO_Manifold_Enabled : ARRAY[1..GVL_CONSTANTS.C_MAX_MANIFOLDS] OF BOOL;
    VO_Heating_Degraded : BOOL;
END_VAR
VAR
    L_i : INT;
    L_j : INT;
    L_Used : REAL;
    L_Selected : ARRAY[1..GVL_CONSTANTS.C_MAX_MANIFOLDS] OF BOOL;
    L_MaxPriority : INT;
    L_CurrentPriority : INT;
END_VAR

VO_Heating_Degraded := FALSE;

// STEP 1: Allowed
FOR L_i := 1 TO GVL_CONSTANTS.C_MAX_MANIFOLDS DO
    VO_Manifold_Allowed[L_i] := TRUE;

    IF NOT VI_Manifold_Pump_In_Service[L_i] THEN
        VO_Manifold_Allowed[L_i] := FALSE;
    END_IF;

    IF VI_Manifold_Pressure_Fault[L_i] THEN
        VO_Manifold_Allowed[L_i] := FALSE;
    END_IF;

    IF VI_Manifold_Current_Fault[L_i] THEN
        VO_Manifold_Allowed[L_i] := FALSE;
    END_IF;

    IF NOT VO_Manifold_Allowed[L_i] THEN
        VO_Heating_Degraded := TRUE;
    END_IF;
END_FOR;

// STEP 2: find max priority
L_MaxPriority := 0;
FOR L_i := 1 TO GVL_CONSTANTS.C_MAX_MANIFOLDS DO
    IF VI_Manifold_Priority[L_i] > L_MaxPriority THEN
        L_MaxPriority := VI_Manifold_Priority[L_i];
    END_IF;
END_FOR;

// STEP 3: allocation by priority + budget
FOR L_i := 1 TO GVL_CONSTANTS.C_MAX_MANIFOLDS DO
    VO_Manifold_Enabled[L_i] := FALSE;
END_FOR;

L_Used := 0.0;

FOR L_CurrentPriority := L_MaxPriority TO 1 BY -1 DO

    FOR L_i := 1 TO GVL_CONSTANTS.C_MAX_MANIFOLDS DO

        IF (VI_Manifold_Priority[L_i] = L_CurrentPriority) AND VO_Manifold_Allowed[L_i] THEN

            IF (L_Used + VI_Manifold_Thermal_Weight[L_i]) <= VI_Max_Thermal_Budget THEN
                VO_Manifold_Enabled[L_i] := TRUE;
                L_Used := L_Used + VI_Manifold_Thermal_Weight[L_i];
            END_IF;

        END_IF;

    END_FOR;

END_FOR;
END_FUNCTION_BLOCK

(* ---- FB_Heating_Diagnostics.st ---- *)
FUNCTION_BLOCK FB_Heating_Diagnostics
VAR_INPUT
    VI_System_Time_MS : UDINT;
END_VAR
VAR
    fbDiagEventManager : FB_Diagnostics_Event_Manager;
    L_i : INT;
    L_Any_Heating_Device_Failed : BOOL;
    L_Critical_Fault : BOOL;
    L_Device_Text : STRING(200);
    L_Critical_Text : STRING(200);
    L_Temp_Text : STRING(200);
    L_Add_Text : STRING(80);
END_VAR

GVL_STATUS.G_Diagnostics.Backup_Pump_Out_Of_Service := NOT GVL_CONFIG.G_Backup_Circulation_Pump_In_Service;
GVL_STATUS.G_Diagnostics.Electric_Heater_Out_Of_Service := NOT GVL_CONFIG.G_Electric_Heater_In_Service;

L_Any_Heating_Device_Failed := FALSE;
L_Device_Text := '';
L_Critical_Text := '';
L_Temp_Text := '';

IF NOT GVL_CONFIG.G_Backup_Circulation_Pump_In_Service THEN
    L_Any_Heating_Device_Failed := TRUE;
    L_Add_Text := 'backup pump out of service';
    IF LEN(L_Device_Text) = 0 THEN
        L_Device_Text := L_Add_Text;
    ELSIF (LEN(L_Device_Text) + LEN(L_Add_Text) + 2) < 200 THEN
        L_Device_Text := CONCAT(L_Device_Text, CONCAT('; ', L_Add_Text));
    END_IF;
END_IF;

IF NOT GVL_CONFIG.G_Electric_Heater_In_Service THEN
    L_Any_Heating_Device_Failed := TRUE;
    L_Add_Text := 'electric heater out of service';
    IF LEN(L_Device_Text) = 0 THEN
        L_Device_Text := L_Add_Text;
    ELSIF (LEN(L_Device_Text) + LEN(L_Add_Text) + 2) < 200 THEN
        L_Device_Text := CONCAT(L_Device_Text, CONCAT('; ', L_Add_Text));
    END_IF;
END_IF;

fbDiagEventManager(VI_Code := GVL_CONFIG.ERR_BACKUP_PUMP_OUT_OF_SERVICE, VI_Severity := 2, VI_Active := NOT GVL_CONFIG.G_Backup_Circulation_Pump_In_Service, VI_Timestamp := VI_System_Time_MS, VI_Source := 400, VIO_Events := GVL_STATUS.G_Diagnostics_Events, VIO_Count := GVL_STATUS.G_Diagnostics_Count);
fbDiagEventManager(VI_Code := GVL_CONFIG.ERR_ELECTRIC_HEATER_OUT_OF_SERVICE, VI_Severity := 2, VI_Active := NOT GVL_CONFIG.G_Electric_Heater_In_Service, VI_Timestamp := VI_System_Time_MS, VI_Source := 401, VIO_Events := GVL_STATUS.G_Diagnostics_Events, VIO_Count := GVL_STATUS.G_Diagnostics_Count);

FOR L_i := 1 TO GVL_CONSTANTS.C_MAX_MANIFOLDS DO
    GVL_STATUS.G_Diagnostics.Manifold_Pump_Out_Of_Service[L_i] := NOT GVL_CONFIG.G_Manifold_Pump_In_Service[L_i];

    IF NOT GVL_CONFIG.G_Manifold_Pump_In_Service[L_i] THEN
        L_Any_Heating_Device_Failed := TRUE;
        L_Add_Text := CONCAT('manifold pump OOS #', INT_TO_STRING(L_i));
        IF LEN(L_Device_Text) = 0 THEN
            L_Device_Text := L_Add_Text;
        ELSIF (LEN(L_Device_Text) + LEN(L_Add_Text) + 2) < 200 THEN
            L_Device_Text := CONCAT(L_Device_Text, CONCAT('; ', L_Add_Text));
        END_IF;
    END_IF;

    fbDiagEventManager(VI_Code := GVL_CONFIG.ERR_MANIFOLD_PUMP_OUT_OF_SERVICE, VI_Severity := 2, VI_Active := NOT GVL_CONFIG.G_Manifold_Pump_In_Service[L_i], VI_Timestamp := VI_System_Time_MS, VI_Source := 410 + L_i, VIO_Events := GVL_STATUS.G_Diagnostics_Events, VIO_Count := GVL_STATUS.G_Diagnostics_Count);
END_FOR;

GVL_STATUS.G_Diagnostics.DHW_Heating_Pump_Out_Of_Service := NOT GVL_CONFIG.G_DHW_Heating_Pump_In_Service;
GVL_STATUS.G_Diagnostics.DHW_Circ_Pump_Out_Of_Service := NOT GVL_CONFIG.G_DHW_Circ_Pump_In_Service;

IF NOT GVL_CONFIG.G_DHW_Heating_Pump_In_Service THEN
    L_Any_Heating_Device_Failed := TRUE;
    L_Add_Text := 'DHW heating pump out of service';
    IF LEN(L_Device_Text) = 0 THEN
        L_Device_Text := L_Add_Text;
    ELSIF (LEN(L_Device_Text) + LEN(L_Add_Text) + 2) < 200 THEN
        L_Device_Text := CONCAT(L_Device_Text, CONCAT('; ', L_Add_Text));
    END_IF;
END_IF;

IF NOT GVL_CONFIG.G_DHW_Circ_Pump_In_Service THEN
    L_Any_Heating_Device_Failed := TRUE;
    L_Add_Text := 'DHW circ pump out of service';
    IF LEN(L_Device_Text) = 0 THEN
        L_Device_Text := L_Add_Text;
    ELSIF (LEN(L_Device_Text) + LEN(L_Add_Text) + 2) < 200 THEN
        L_Device_Text := CONCAT(L_Device_Text, CONCAT('; ', L_Add_Text));
    END_IF;
END_IF;

fbDiagEventManager(VI_Code := GVL_CONFIG.ERR_DHW_HEATING_PUMP_OUT_OF_SERVICE, VI_Severity := 2, VI_Active := NOT GVL_CONFIG.G_DHW_Heating_Pump_In_Service, VI_Timestamp := VI_System_Time_MS, VI_Source := 420, VIO_Events := GVL_STATUS.G_Diagnostics_Events, VIO_Count := GVL_STATUS.G_Diagnostics_Count);
fbDiagEventManager(VI_Code := GVL_CONFIG.ERR_DHW_CIRC_PUMP_OUT_OF_SERVICE, VI_Severity := 2, VI_Active := NOT GVL_CONFIG.G_DHW_Circ_Pump_In_Service, VI_Timestamp := VI_System_Time_MS, VI_Source := 421, VIO_Events := GVL_STATUS.G_Diagnostics_Events, VIO_Count := GVL_STATUS.G_Diagnostics_Count);

L_Critical_Fault := GVL_STATE.G_Freeze_Hardware_Failed;
IF L_Critical_Fault THEN
    L_Critical_Text := 'Freeze hardware critical fault';
END_IF;

fbDiagEventManager(VI_Code := GVL_CONFIG.ERR_FREEZE_HARDWARE_FAILED, VI_Severity := 4, VI_Active := GVL_STATE.G_Freeze_Hardware_Failed, VI_Timestamp := VI_System_Time_MS, VI_Source := 430, VIO_Events := GVL_STATUS.G_Diagnostics_Events, VIO_Count := GVL_STATUS.G_Diagnostics_Count);

GVL_STATE.G_Heating_Subsystem_Degraded := GVL_STATE.G_Heating_Subsystem_Degraded OR L_Any_Heating_Device_Failed;
GVL_STATE.G_Freeze_Hardware_Degraded := GVL_STATE.G_Freeze_Hardware_Degraded OR L_Any_Heating_Device_Failed;
GVL_STATUS.G_Diagnostics.Freeze_Hardware_Event_Pending := GVL_STATUS.G_Diagnostics.Freeze_Hardware_Event_Pending OR L_Critical_Fault OR L_Any_Heating_Device_Failed;

IF L_Critical_Fault AND L_Any_Heating_Device_Failed THEN
    L_Temp_Text := CONCAT(L_Critical_Text, '; ');
    IF (LEN(L_Temp_Text) + LEN(L_Device_Text)) < 200 THEN
        L_Temp_Text := CONCAT(L_Temp_Text, L_Device_Text);
    END_IF;
    GVL_STATUS.G_Diagnostics.Freeze_Hardware_Event_Text := L_Temp_Text;
ELSIF L_Critical_Fault THEN
    GVL_STATUS.G_Diagnostics.Freeze_Hardware_Event_Text := L_Critical_Text;
ELSIF L_Any_Heating_Device_Failed THEN
    GVL_STATUS.G_Diagnostics.Freeze_Hardware_Event_Text := L_Device_Text;
END_IF;

END_FUNCTION_BLOCK
// >>> BULK_SYNC_ANCHOR: FB_Heating_Diagnostics <<<

(* ---- FB_Heating_Local_Context.st ---- *)
FUNCTION_BLOCK FB_Heating_Local_Context
VAR_INPUT
    VI_System_Time_MS : UDINT;
    VI_Heating_Emergency_Stop : BOOL;
    VI_Heating_Gas_Safety_Stop : BOOL;
    VI_DHW_Block : BOOL;
    VI_Freeze_Request : BOOL;
    VI_Preheat_Request : BOOL;
    VI_DHW_Heating_Pump_Feedback : BOOL;
    VI_Policy_Target_Adjustment : REAL;
    VI_Boiler_Modulation_Raw : ARRAY[1..GVL_CONSTANTS.C_MAX_BOILERS] OF INT;
END_VAR
VAR_OUTPUT
    VO_Boiler_Modulation_REAL : ARRAY[1..GVL_CONSTANTS.C_MAX_BOILERS] OF REAL;
    VO_Heating_Emergency_Stop : BOOL;
    VO_Heating_Gas_Safety_Stop : BOOL;
    VO_Heating_DHW_Demand : BOOL;
    VO_Target_Temperature : REAL;
    VO_Local_Mode : INT;
END_VAR
VAR
    L_Last_Mode : INT := 0;
    L_Mode_Hold_Timer : FB_System_Timer;
    L_i : INT;
END_VAR

FOR L_i := 1 TO GVL_CONSTANTS.C_MAX_BOILERS DO
    VO_Boiler_Modulation_REAL[L_i] := TO_REAL(VI_Boiler_Modulation_Raw[L_i]);
END_FOR;

VO_Heating_Emergency_Stop := VI_Heating_Emergency_Stop;
VO_Heating_Gas_Safety_Stop := VI_Heating_Gas_Safety_Stop;
VO_Heating_DHW_Demand := VI_DHW_Heating_Pump_Feedback;

IF VO_Heating_Emergency_Stop THEN
    VO_Heating_Gas_Safety_Stop := FALSE;
    VO_Heating_DHW_Demand := FALSE;
ELSIF VO_Heating_Gas_Safety_Stop THEN
    VO_Heating_DHW_Demand := FALSE;
ELSIF VI_DHW_Block THEN
    VO_Heating_DHW_Demand := FALSE;
END_IF;

L_Mode_Hold_Timer(IN := TRUE, PT := T#30s, VI_System_Time_MS := VI_System_Time_MS);

IF L_Mode_Hold_Timer.Q THEN
    IF VI_Freeze_Request THEN L_Last_Mode := 2;
    ELSIF VI_Preheat_Request THEN L_Last_Mode := 1;
    ELSE L_Last_Mode := 0;
    END_IF;
END_IF;

CASE L_Last_Mode OF
    2: VO_Target_Temperature := 5.0;
    1: VO_Target_Temperature := 22.0;
    ELSE VO_Target_Temperature := 20.0;
END_CASE;

VO_Target_Temperature := VO_Target_Temperature + VI_Policy_Target_Adjustment;
IF VO_Target_Temperature < 5.0 THEN VO_Target_Temperature := 5.0;
ELSIF VO_Target_Temperature > 26.0 THEN VO_Target_Temperature := 26.0;
END_IF;

VO_Local_Mode := L_Last_Mode;

END_FUNCTION_BLOCK
// >>> BULK_SYNC_ANCHOR: FB_Heating_Local_Context <<<

(* ---- FB_Heating_Maintenance_Gating.st ---- *)
FUNCTION_BLOCK FB_Heating_Maintenance_Gating
VAR
    L_i : INT;
END_VAR

// Extracted candidate from PRG_Heating S4.
// Not connected yet.
// Donor logic remains in PRG_Heating until all extracted candidates are prepared.

IF NOT GVL_CONFIG.G_Backup_Circulation_Pump_In_Service THEN
    GVL_STATE.G_Backup_Circulation_Pump := FALSE;
END_IF;
IF NOT GVL_CONFIG.G_Electric_Heater_In_Service THEN
    GVL_STATE.G_Electric_Heater_Enable := FALSE;
END_IF;
FOR L_i := 1 TO GVL_CONSTANTS.C_MAX_MANIFOLDS DO
    IF NOT GVL_CONFIG.G_Manifold_Pump_In_Service[L_i] THEN
        GVL_STATE.G_Manifold_Pumps[L_i] := FALSE;
    END_IF;
END_FOR;
IF NOT GVL_CONFIG.G_DHW_Heating_Pump_In_Service THEN
    GVL_STATE.G_DHW_Heating_Pump := FALSE;
END_IF;
IF NOT GVL_CONFIG.G_DHW_Circ_Pump_In_Service THEN
    GVL_STATE.G_DHW_Circ_Pump := FALSE;
END_IF;

END_FUNCTION_BLOCK
// >>> BULK_SYNC_ANCHOR: FB_Heating_Maintenance_Gating <<<

(* ---- FB_Heating_Predictive_Controller.st ---- *)
FUNCTION_BLOCK FB_Heating_Predictive_Controller
VAR
    L_i : INT;
    L_Time_To_Heat : UDINT;
    L_Time_To_Comfort : UDINT;
    L_Now_TOD : UDINT;
END_VAR

L_Now_TOD := GVL_TIME_SERVICE.G_Time_Of_Day_MS;

FOR L_i := 1 TO GVL_CONSTANTS.C_MAX_ZONES DO

    L_Time_To_Heat := GVL_HEATING_POLICY.G_Zone_Time_To_Heat_MS[L_i];
    L_Time_To_Comfort := GVL_HEATING_POLICY.G_Zone_Comfort_Time_MS[L_i];

    // predictive preheat decision
    IF GVL_HEATING_POLICY.G_Zone_Schedule_Enabled[L_i] THEN

        IF L_Time_To_Comfort > L_Now_TOD THEN
            IF (L_Time_To_Comfort - L_Now_TOD) <= L_Time_To_Heat THEN
                GVL_HEATING_POLICY.G_Zone_Preheat_Needed[L_i] := TRUE;
            ELSE
                GVL_HEATING_POLICY.G_Zone_Preheat_Needed[L_i] := FALSE;
            END_IF;
        END_IF;

    END_IF;

    // overshoot prevention
    IF GVL_HEATING_POLICY.G_Zone_Predicted_Temp_30m[L_i] > GVL_STATE.G_Target_Temperature THEN
        GVL_HEATING_POLICY.G_Zone_Thermal_Demand[L_i] :=
            GVL_HEATING_POLICY.G_Zone_Thermal_Demand[L_i] * 0.5;
    END_IF;

    // confidence gating
    IF GVL_HEATING_POLICY.G_Zone_Thermal_Model_Confidence[L_i] < 0.1 THEN
        GVL_HEATING_POLICY.G_Zone_Preheat_Needed[L_i] := FALSE;
    END_IF;

END_FOR;

END_FUNCTION_BLOCK

(* ---- FB_Heating_RootCause_Diagnostics.st ---- *)
FUNCTION_BLOCK FB_Heating_RootCause_Diagnostics
VAR_INPUT
    VI_Zone_Valves : ARRAY[1..GVL_CONSTANTS.C_MAX_HEATING_CIRCUITS] OF BOOL;
END_VAR
VAR
    fbRootCause : FB_Diagnostics_RootCause;
    fbRootDemandMap : FB_Heating_Demand_Map;
    L_Root_Demand_Map : ARRAY[1..GVL_CONSTANTS.C_MAX_MANIFOLDS] OF BOOL;
END_VAR

// Extracted candidate from PRG_Heating S7.
// Not connected yet.
// Donor logic remains in PRG_Heating until all extracted candidates are prepared.

fbRootDemandMap(
    VI_Zone_Valves := VI_Zone_Valves,
    VI_Zone_Configs := GVL_CONFIG.G_HMI_FloorHeating_Configs,
    VO_Manifold_Demand_Map => L_Root_Demand_Map
);

fbRootCause(
    VI_Emergency_Stop := GVL_STATE.G_Safety_Emergency_Stop,
    VI_Gas_Safety := GVL_STATE.G_Safety_Gas_Latched,
    VI_IO_Failsafe := GVL_STATE.G_Heating_IO_Fault,
    VI_Boiler_OT_Online := GVL_STATE.G_Boiler_OT_Online,
    VI_Boiler_Error := GVL_STATE.G_Boiler_Error,
    VI_Boiler_Flame := GVL_STATE.G_Boiler_Flame,
    VI_Manifold_Pumps := GVL_STATE.G_Manifold_Pumps,
    VI_Manifold_Valves := GVL_STATE.G_Manifold_Valves,
    VI_Sensor_Error := GVL_STATE.G_Heating_Sensor_Fault,
    VI_Supply_Temps := GVL_STATE.G_Manifold_T_Supply,
    VI_Target_Supply := GVL_CONFIG.G_Heating_Config.Target_Floor_Temp,
    VI_Demand_Map := L_Root_Demand_Map
);

GVL_STATE.G_Heating_RootCause := fbRootCause.VO_RootCause;
GVL_STATE.G_Heating_RootConfidence := fbRootCause.VO_Confidence;

END_FUNCTION_BLOCK
// >>> BULK_SYNC_ANCHOR: FB_Heating_RootCause_Diagnostics <<<

(* ---- FB_Heating_Schedule_Preheat.st ---- *)
FUNCTION_BLOCK FB_Heating_Schedule_Preheat
VAR_INPUT
    VI_System_Time_MS : UDINT;
    VI_Time_Of_Day_MS : UDINT;
    VI_Day_Of_Week : INT; // 1=Mon ... 7=Sun
    VI_Enable : BOOL;
END_VAR

VAR
    L_i : INT;
    L_e : INT;
    L_Event : ST_Heating_Schedule_Event;
    L_Time_To_Comfort_MS : UDINT;
    L_Adjustment : REAL;
    L_Max_Boost : REAL;
    L_Active : BOOL;

    L_Learn_Window_MS : UDINT := 300000;
    L_Learn_Cooldown_MS : UDINT := 900000;
    L_Cold_Confirm : ARRAY[1..GVL_CONSTANTS.C_MAX_ZONES, 1..3] OF INT;
    L_Hot_Confirm : ARRAY[1..GVL_CONSTANTS.C_MAX_ZONES, 1..3] OF INT;
    L_Last_Learn_MS : ARRAY[1..GVL_CONSTANTS.C_MAX_ZONES, 1..3] OF UDINT;
    L_Elapsed_MS : UDINT;
END_VAR

IF NOT VI_Enable THEN
    FOR L_i := 1 TO GVL_CONSTANTS.C_MAX_ZONES DO
        GVL_HEATING_POLICY.G_Zone_Schedule_Preheat_Active[L_i] := FALSE;
    END_FOR;
    RETURN;
END_IF;

FOR L_i := 1 TO GVL_CONSTANTS.C_MAX_ZONES DO
    L_Active := FALSE;
    L_Max_Boost := 0.0;

    FOR L_e := 1 TO 3 DO
        L_Event := GVL_HEATING_POLICY_CONFIG.G_Zone_Schedule[L_i, L_e];

        IF L_Event.Enabled THEN
            IF (L_Event.Weekday_Mask AND SHL(1, VI_Day_Of_Week - 1)) <> 0 THEN

                IF L_Event.Comfort_Time_MS >= VI_Time_Of_Day_MS THEN
                    L_Time_To_Comfort_MS := L_Event.Comfort_Time_MS - VI_Time_Of_Day_MS;
                ELSE
                    L_Time_To_Comfort_MS := (86400000 - VI_Time_Of_Day_MS) + L_Event.Comfort_Time_MS;
                END_IF;

                IF L_Event.Adaptive_Enabled THEN
                    IF GVL_HEATING_POLICY.G_Zone_Schedule_Learned_Offset_MS[L_i, L_e] > L_Event.Adaptive_Max_Offset_MS THEN
                        GVL_HEATING_POLICY.G_Zone_Schedule_Learned_Offset_MS[L_i, L_e] := L_Event.Adaptive_Max_Offset_MS;
                    END_IF;
                    L_Time_To_Comfort_MS := L_Time_To_Comfort_MS + GVL_HEATING_POLICY.G_Zone_Schedule_Learned_Offset_MS[L_i, L_e];
                END_IF;

                IF (GVL_HEATING_POLICY.G_Zone_Time_To_Heat_MS[L_i] >= L_Time_To_Comfort_MS)
                   AND (GVL_HEATING_POLICY.G_Zone_Time_To_Heat_MS[L_i] > 0) THEN

                    IF L_Event.Preheat_Boost > L_Max_Boost THEN
                        L_Max_Boost := L_Event.Preheat_Boost;
                    END_IF;

                    L_Active := TRUE;
                END_IF;

                IF L_Event.Adaptive_Enabled THEN
                    IF L_Time_To_Comfort_MS < L_Learn_Window_MS THEN

                        IF GVL_HEATING_POLICY.G_Zone_Thermal_Demand[L_i] > 1.0 THEN
                            L_Cold_Confirm[L_i, L_e] := L_Cold_Confirm[L_i, L_e] + 1;
                            L_Hot_Confirm[L_i, L_e] := 0;
                        ELSIF GVL_HEATING_POLICY.G_Zone_Thermal_Demand[L_i] < -0.5 THEN
                            L_Hot_Confirm[L_i, L_e] := L_Hot_Confirm[L_i, L_e] + 1;
                            L_Cold_Confirm[L_i, L_e] := 0;
                        ELSE
                            L_Cold_Confirm[L_i, L_e] := 0;
                            L_Hot_Confirm[L_i, L_e] := 0;
                        END_IF;

                        // UDINT wrap-safe elapsed time; unsigned subtraction is valid modulo 2^32.
                        L_Elapsed_MS := VI_System_Time_MS - L_Last_Learn_MS[L_i, L_e];

                        IF L_Elapsed_MS >= L_Learn_Cooldown_MS THEN

                            IF L_Cold_Confirm[L_i, L_e] >= 2 THEN
                                IF GVL_HEATING_POLICY.G_Zone_Schedule_Learned_Offset_MS[L_i, L_e] < L_Event.Adaptive_Max_Offset_MS THEN
                                    GVL_HEATING_POLICY.G_Zone_Schedule_Learned_Offset_MS[L_i, L_e] :=
                                        GVL_HEATING_POLICY.G_Zone_Schedule_Learned_Offset_MS[L_i, L_e] + L_Event.Adaptive_Step_MS;
                                    IF GVL_HEATING_POLICY.G_Zone_Schedule_Learned_Offset_MS[L_i, L_e] > L_Event.Adaptive_Max_Offset_MS THEN
                                        GVL_HEATING_POLICY.G_Zone_Schedule_Learned_Offset_MS[L_i, L_e] := L_Event.Adaptive_Max_Offset_MS;
                                    END_IF;
                                    L_Last_Learn_MS[L_i, L_e] := VI_System_Time_MS;
                                END_IF;
                                L_Cold_Confirm[L_i, L_e] := 0;
                            END_IF;

                            IF L_Hot_Confirm[L_i, L_e] >= 2 THEN
                                IF GVL_HEATING_POLICY.G_Zone_Schedule_Learned_Offset_MS[L_i, L_e] > L_Event.Adaptive_Step_MS THEN
                                    GVL_HEATING_POLICY.G_Zone_Schedule_Learned_Offset_MS[L_i, L_e] :=
                                        GVL_HEATING_POLICY.G_Zone_Schedule_Learned_Offset_MS[L_i, L_e] - L_Event.Adaptive_Step_MS;
                                ELSE
                                    GVL_HEATING_POLICY.G_Zone_Schedule_Learned_Offset_MS[L_i, L_e] := 0;
                                END_IF;
                                L_Last_Learn_MS[L_i, L_e] := VI_System_Time_MS;
                                L_Hot_Confirm[L_i, L_e] := 0;
                            END_IF;

                        END_IF;
                    ELSE
                        L_Cold_Confirm[L_i, L_e] := 0;
                        L_Hot_Confirm[L_i, L_e] := 0;
                    END_IF;
                END_IF;

            END_IF;
        END_IF;
    END_FOR;

    L_Adjustment := GVL_HEATING_POLICY.G_Zone_Target_Adjustment[L_i];

    IF L_Active AND (L_Adjustment < L_Max_Boost) THEN
        L_Adjustment := L_Max_Boost;
    END_IF;

    IF L_Adjustment > 1.0 THEN
        L_Adjustment := 1.0;
    ELSIF L_Adjustment < -1.0 THEN
        L_Adjustment := -1.0;
    END_IF;

    GVL_HEATING_POLICY.G_Zone_Target_Adjustment[L_i] := L_Adjustment;
    GVL_HEATING_POLICY.G_Zone_Schedule_Preheat_Active[L_i] := L_Active;
END_FOR;

END_FUNCTION_BLOCK

(* ---- FB_NVRAM_Manager.st ---- *)
FUNCTION_BLOCK FB_NVRAM_Manager
VAR_INPUT
    VI_Command                  : BYTE; // 1=WRITE (READ not implemented)
    VI_Offset                   : UDINT; // Смещение в байтах
    VI_DataRef                  : REFERENCE TO BYTE;
    VI_DataSize                 : UDINT; // КРИТИЧНО: используем этот размер вместо SIZEOF
    VI_System_Time_MS           : UDINT;
    VI_Operator_ID              : STRING(10);
    VI_IsActivePLC              : BOOL;
    VI_TwoPersonConfirmation    : BOOL;
END_VAR
VAR_OUTPUT
    VO_Done                     : BOOL;
    VO_Error                    : BOOL;
    VO_ErrorID                  : UDINT;
    // VO_ReadDataRef removed (REFERENCE TO not allowed in output)
    VO_HMI_Status_Message       : STRING(200);
END_VAR
VAR
    L_prev_Command              : BYTE;
    L_cmd_rising                : BOOL;
    L_i                         : UDINT;
    L_Data_Changed              : BOOL; // Флаг изменения данных
    L_pData                      : POINTER TO BYTE;
END_VAR
VAR CONSTANT
    C_MAX_NVRAM_SIZE            : UDINT := 12800;
END_VAR

// Детекция фронта команды
L_cmd_rising := (VI_Command <> 0) AND (L_prev_Command = 0);
L_prev_Command := VI_Command;

IF L_cmd_rising THEN
    VO_Done := FALSE;
    VO_Error := FALSE;
    VO_ErrorID := 0;
    VO_HMI_Status_Message := '';

    // Валидация смещения
    IF VI_Offset >= C_MAX_NVRAM_SIZE THEN
        VO_Error := TRUE;
        VO_ErrorID := 16#1501;
        VO_HMI_Status_Message := 'NVRAM: Неверное смещение';
        VO_Done := TRUE;
        RETURN;
    END_IF;

    // Валидация указателя
    IF NOT __ISVALIDREF(VI_DataRef) THEN
        VO_Error := TRUE;
        VO_ErrorID := 16#150A;
        VO_HMI_Status_Message := 'NVRAM: Недействительная ссылка на данные';
        VO_Done := TRUE;
        RETURN;
    END_IF;

    L_pData := ADR(VI_DataRef);

    IF (VI_Offset + VI_DataSize) > C_MAX_NVRAM_SIZE THEN
        VO_Error := TRUE;
        VO_ErrorID := 16#150B;
        VO_HMI_Status_Message := 'NVRAM: Размер данных превышает доступный объем';
        VO_Done := TRUE;
        RETURN;
    END_IF;

    IF VI_Command = 2 THEN
    VO_Error := TRUE;
    VO_ErrorID := 16#150D;
    VO_HMI_Status_Message := 'NVRAM: READ not implemented';
    VO_Done := TRUE;
    RETURN;
END_IF;

IF VI_Command = 1 THEN // ЗАПИСЬ (WRITE)
        IF NOT VI_IsActivePLC THEN
            VO_Error := TRUE;
            VO_ErrorID := 16#1509;
            VO_HMI_Status_Message := 'NVRAM: Запись запрещена (STANDBY)';
        ELSE
            // Проверка на изменение данных перед записью
            L_Data_Changed := FALSE;
            FOR L_i := 0 TO VI_DataSize - 1 DO
                IF GVL_Retain.G_NVRAM_Data[VI_Offset + L_i] <> L_pData[L_i] THEN
                    L_Data_Changed := TRUE;
                    EXIT;
                END_IF;
            END_FOR;

            IF L_Data_Changed THEN
                // Безопасное копирование (WRITE)
                FOR L_i := 0 TO VI_DataSize - 1 DO
                    GVL_Retain.G_NVRAM_Data[VI_Offset + L_i] := L_pData[L_i];
                END_FOR;
                VO_HMI_Status_Message := 'NVRAM: Данные успешно сохранены в RETAIN';
            ELSE
                VO_HMI_Status_Message := 'NVRAM: Данные не изменились, запись пропущена';
            END_IF;
        END_IF;
        VO_Done := TRUE;
    END_IF;
END_IF;

IF VI_Command = 0 THEN
    VO_Done := FALSE;
END_IF;
// >>> BULK_SYNC_ANCHOR: FB_NVRAM_Manager <<<
END_FUNCTION_BLOCK

(* ---- FB_PLC_Heartbeat.st ---- *)
FUNCTION_BLOCK FB_PLC_Heartbeat
VAR_INPUT
    VI_Local_ID : BYTE; // Идентификатор данного ПЛК (1 - ПЛК А, 2 - ПЛК B)
    VI_System_Time : UDINT; // Текущее системное время (мс)
    VI_Remote_Pulse : BOOL; // Сигнал пульса от партнерского ПЛК
    VI_Remote_Is_Active : BOOL; // Статус активности партнерского ПЛК (ТЗ 8.3)
    VI_Gateway_Ping_OK : BOOL; // Флаг доступности сетевого шлюза (ТЗ 8.3)
END_VAR
VAR_OUTPUT
    VO_Is_Active : BOOL; // Выход: Данный ПЛК является ведущим (Active)
    VO_RTT_MS : UDINT; // Текущая задержка связи между ПЛК (Round Trip Time)
    VO_Loss_Count : UDINT; // Счетчик потерь пакетов связи (ТЗ 8.4)
    VO_Max_RTT : UDINT; // Максимальная зафиксированная задержка связи
END_VAR
VAR
    L_Last_Pulse : BOOL; // Предыдущее состояние сигнала пульса
    L_Last_Pulse_Time : UDINT; // Время последнего изменения сигнала пульса
    L_Timeout : UDINT := 500; // Порог таймаута связи (500 мс по ТЗ 8.1)
    L_Pulse_Send_Time : UDINT; // Время отправки собственного пульса
    L_Last_Loss_Time : UDINT; // Время последней фиксации потери связи
    L_Elapsed_Time : UDINT;
END_VAR

// Вспомогательная функция для безопасного вычисления разницы времени
L_Elapsed_Time := (VI_System_Time - L_Last_Pulse_Time);

// 1. Мониторинг "сердцебиения" и расчет сетевых задержек (ТЗ 8.4)
IF VI_Remote_Pulse <> L_Last_Pulse THEN
    // Вычисляем время между изменениями сигнала
    VO_RTT_MS := L_Elapsed_Time;
    // Фиксируем пиковые задержки для диагностики сети
    IF VO_RTT_MS > VO_Max_RTT THEN VO_Max_RTT := VO_RTT_MS; END_IF;
    L_Last_Pulse := VI_Remote_Pulse;
    L_Last_Pulse_Time := VI_System_Time;
    L_Elapsed_Time := 0; // Сбрасываем после обновления
END_IF;

// Подсчет статистики потерь связи (ТЗ 8.4)
IF L_Elapsed_Time > L_Timeout THEN
    IF (VI_System_Time - L_Last_Loss_Time) >= 1000 THEN
        VO_Loss_Count := VO_Loss_Count + 1;
        L_Last_Loss_Time := VI_System_Time;
    END_IF;
ELSE
    L_Last_Loss_Time := VI_System_Time;
END_IF;

// 2. Логика определения роли (Active/Standby) и предотвращение Split-Brain (ТЗ 8.3)
// Уровень 1: Проверка наличия связи с партнером
IF L_Elapsed_Time < L_Timeout THEN
    // Связь есть: Договариваемся о ролях на основе приоритета ID
    IF VI_Local_ID = 1 THEN
        VO_Is_Active := TRUE; // ПЛК А всегда активен при наличии связи
    ELSE
        VO_Is_Active := NOT VI_Remote_Is_Active; // ПЛК B активен только если А не активен
    END_IF;
ELSE
    // Связи нет: Пытаемся определить, кто из нас "живее"
    // Уровень 3: Если связи с партнером нет, проверяем доступность внешнего шлюза
    IF VI_Local_ID = 1 THEN
        // ПЛК А становится активным всегда при потере связи с партнером (fallback)
        VO_Is_Active := TRUE;
    ELSE
        // ПЛК B ждет таймаут удержания роли (2 секунды), прежде чем стать активным
        IF L_Elapsed_Time >= 2000 THEN
            // ПЛК B берет управление если он видит шлюз, а связи с А нет.
            // Если шлюз недоступен, B ждет дольше (fallback).
            IF VI_Gateway_Ping_OK THEN
                VO_Is_Active := TRUE;
            ELSIF L_Elapsed_Time >= 5000 THEN
                VO_Is_Active := TRUE; // Fallback: ПЛК А мертв и шлюз мертв
            ELSE
                VO_Is_Active := FALSE;
            END_IF;
        ELSE
            VO_Is_Active := FALSE;
        END_IF;
    END_IF;
END_IF;
END_FUNCTION_BLOCK

(* ---- FB_Random_Generator.st ---- *)
FUNCTION_BLOCK FB_Random_Generator
VAR
    L_seed : UDINT := 1;
    L_Is_Seeded : BOOL := FALSE;
END_VAR
VAR CONSTANT
    C_LCG_MULTIPLIER : UDINT := 1664525;
    C_LCG_INCREMENT  : UDINT := 1013904223;
    C_LCG_MODULUS    : LREAL := 4294967296.0;
END_VAR

METHOD Seed : BOOL
VAR_INPUT
    VI_Seed_Value : UDINT;
END_VAR
L_seed := VI_Seed_Value;
L_Is_Seeded := TRUE;
Seed := TRUE;
END_METHOD

METHOD Random_Int_Range : UDINT
VAR_INPUT
    VI_min : UDINT;
    VI_max : UDINT;
    VI_System_Time_MS : UDINT; // Для автоматического сидирования
END_VAR
VAR
    L_range : UDINT;
    L_rand_factor : LREAL;
END_VAR

IF NOT L_Is_Seeded AND VI_System_Time_MS > 0 THEN
    L_seed := VI_System_Time_MS;
    L_Is_Seeded := TRUE;
END_IF;

L_seed := (C_LCG_MULTIPLIER * L_seed) + C_LCG_INCREMENT;

IF VI_max > VI_min THEN
        L_range := VI_max - VI_min;
        // Используем LREAL для точности и исключения выхода за границу
        L_rand_factor := TO_LREAL(L_seed) / C_LCG_MODULUS;
        Random_Int_Range := VI_min + TO_UDINT(L_rand_factor * TO_LREAL(L_range + 1));

        // Финальная защита от переполнения
        IF Random_Int_Range > VI_max THEN
            Random_Int_Range := VI_max;
        END_IF;
    ELSE
        Random_Int_Range := VI_min;
    END_IF;
END_FUNCTION_BLOCK

(* ---- FB_Scenario_Transition_Guard.st ---- *)
FUNCTION_BLOCK FB_Scenario_Transition_Guard
VAR_INPUT
    VI_Current_Scenario : E_SCENARIO_TYPE;
    VI_Target_Scenario  : E_SCENARIO_TYPE;
END_VAR

VAR_OUTPUT
    VO_Transition_Allowed : BOOL;
    VO_Reason             : STRING(120);
END_VAR

VO_Transition_Allowed := TRUE;
VO_Reason := 'OK';

// no-op transition is always allowed
IF VI_Current_Scenario = VI_Target_Scenario THEN
    RETURN;
END_IF;

// emergency can always be entered
IF VI_Target_Scenario = E_SCENARIO_TYPE.SCENARIO_EMERGENCY THEN
    RETURN;
END_IF;

// from NONE, any target is allowed
IF VI_Current_Scenario = E_SCENARIO_TYPE.SCENARIO_NONE THEN
    RETURN;
END_IF;

// emergency exit is restricted
IF VI_Current_Scenario = E_SCENARIO_TYPE.SCENARIO_EMERGENCY THEN
    CASE VI_Target_Scenario OF
        E_SCENARIO_TYPE.SCENARIO_NONE,
        E_SCENARIO_TYPE.SCENARIO_AWAY,
        E_SCENARIO_TYPE.SCENARIO_SLEEP,
        E_SCENARIO_TYPE.SCENARIO_PRESENCE:
            RETURN;
    ELSE
        VO_Transition_Allowed := FALSE;
        VO_Reason := 'Переход из EMERGENCY в данный сценарий запрещён';
        RETURN;
    END_CASE;
END_IF;

// away exit is restricted to safe occupancy contexts
IF VI_Current_Scenario = E_SCENARIO_TYPE.SCENARIO_AWAY THEN
    CASE VI_Target_Scenario OF
        E_SCENARIO_TYPE.SCENARIO_NONE,
        E_SCENARIO_TYPE.SCENARIO_SLEEP,
        E_SCENARIO_TYPE.SCENARIO_PRESENCE,
        E_SCENARIO_TYPE.SCENARIO_EMERGENCY:
            RETURN;
    ELSE
        VO_Transition_Allowed := FALSE;
        VO_Reason := 'Переход из AWAY в данный сценарий запрещён';
        RETURN;
    END_CASE;
END_IF;

// default: allow
RETURN;
// >>> BULK_SYNC_ANCHOR: FB_Scenario_Transition_Guard <<<
END_FUNCTION_BLOCK

(* ---- FB_Sensor_Calibration_Processor.st ---- *)
FUNCTION_BLOCK FB_Sensor_Calibration_Processor
VAR_INPUT
    VI_Raw_Value : REAL;
    VI_Record    : ST_Sensor_Calibration_Record;
END_VAR
VAR_OUTPUT
    VO_Calibrated_Value : REAL;
END_VAR

VO_Calibrated_Value := (VI_Raw_Value * VI_Record.multiplier) + VI_Record.offset;
END_FUNCTION_BLOCK

(* ---- FB_State_Trace_Log.st ---- *)
FUNCTION_BLOCK FB_State_Trace_Log
VAR_INPUT
    VI_System_Time : UDINT;
    VI_Gas_Alarm : BOOL;
    VI_Leak_Alarm : BOOL;
    VI_Pumps : ARRAY[1..4] OF BOOL;
END_VAR
VAR_OUTPUT
    VO_Last_Change_Time : UDINT;
END_VAR
VAR
    L_Last_Gas : BOOL;
    L_Last_Leak : BOOL;
END_VAR

IF (VI_Gas_Alarm <> L_Last_Gas) OR (VI_Leak_Alarm <> L_Last_Leak) THEN
    VO_Last_Change_Time := VI_System_Time;
END_IF;

L_Last_Gas := VI_Gas_Alarm;
L_Last_Leak := VI_Leak_Alarm;
END_FUNCTION_BLOCK

(* ---- FB_System_Alarm_Orchestrator.st ---- *)
// ==============================================================================
// System alarm orchestrator helper
//
// Internal helper for PRG_System.
// Owns FB_Alarm_Manager call and alarm output projection.
// ==============================================================================
FUNCTION_BLOCK FB_System_Alarm_Orchestrator
VAR_INPUT
    VI_First_Fault_Active : BOOL;
    VI_First_Fault_Type : INT;
    VI_First_Fault_Source : INT;
END_VAR

VAR
    fbAlarmManager : FB_Alarm_Manager;
END_VAR

fbAlarmManager(
    VI_System_Time_MS := GVL_STATUS.G_System_Time_MS,
    VI_IsActivePLC := GVL_STATUS.G_Is_Active_PLC,
    VI_Gas_Alarm := GVL_ALARM.G_Gas_Alarm_Active,
    VI_Fire_Alarm := GVL_ALARM.G_Fire_Alarm_Active,
    VI_Flood_Alarm := GVL_ALARM.G_Flood_Alarm_Active,
    VI_Security_Alarm := GVL_ALARM.G_Security_Alarm,
    VI_First_Fault_Active := VI_First_Fault_Active,
    VI_First_Fault_Type := VI_First_Fault_Type,
    VI_First_Fault_Source := VI_First_Fault_Source,
    VI_Boiler_Errors := GVL_STATE.G_Boiler_Error,
    VI_Security_Msg := GVL_STATUS.G_Security_Status_Msg,
    VI_Acknowledge_All := GVL_CONFIG.G_HMI_Ack_Alarms OR GVL_COMMAND.G_Reset_Errors,
    VI_Mute_Siren := GVL_CONFIG.G_HMI_Mute_Alarm,
    VIO_Next_Alarm_ID := GVL_ALARM.G_Next_Alarm_ID,
    VO_Global_Critical => GVL_ALARM.G_Global_Critical,
    VO_Global_Warning => GVL_ALARM.G_Global_Warning,
    VO_Siren_Active => GVL_ALARM.G_Global_Siren,
    VO_Active_Count => GVL_ALARM.G_Active_Alarm_Count,
    VO_Unacked_Count => GVL_ALARM.G_Unacked_Alarm_Count,
    VO_Event_Pulse => GVL_STATUS.G_Diagnostics.Alarm_Event_Pulse,
    VO_Event_Code => GVL_STATUS.G_Diagnostics.Alarm_Event_Code,
    VO_Event_Value => GVL_STATUS.G_Diagnostics.Alarm_Event_Value,
    VO_Alarm_List => GVL_ALARM.G_Alarm_List
);

// >>> BULK_SYNC_ANCHOR: FB_System_Alarm_Orchestrator <<<
END_FUNCTION_BLOCK

(* ---- FB_System_Init.st ---- *)
// ==============================================================================
// System init helper
//
// Internal helper for PRG_System.
// Owns first-boot initialization of RETAIN runtime state.
// ==============================================================================
FUNCTION_BLOCK FB_System_Init
VAR_IN_OUT
    VIO_Local_State : ST_System_State_Snapshot;
    VIO_Remote_State : ST_System_State_Snapshot;
END_VAR

VAR
    L_i : INT;
END_VAR

IF NOT GVL_Retain.G_Initialized THEN
    FOR L_i := 0 TO GVL_CONSTANTS.C_MAX_PRESENCE_HISTORY - 1 DO
        GVL_Retain.G_Presence_History[L_i] := 0;
    END_FOR;

    GVL_Retain.G_History_Write_Idx := 1;
    GVL_Retain.G_History_Total_Events := 0;

    FOR L_i := 1 TO GVL_CONSTANTS.C_MAX_BOILERS DO
        GVL_Retain.G_Boiler_Accumulated_MS[L_i] := 0;
        GVL_Retain.G_Boiler_Work_Seconds[L_i] := 0;
    END_FOR;

    FOR L_i := 1 TO GVL_CONSTANTS.C_MAX_MANIFOLDS DO
        GVL_Retain.G_Valve_Test_Results[L_i] := FALSE;
    END_FOR;

    VIO_Local_State.Version := 0;
    VIO_Remote_State.Version := 0;

    GVL_Retain.G_Initialized := TRUE;
END_IF;

// >>> BULK_SYNC_ANCHOR: FB_System_Init <<<
END_FUNCTION_BLOCK

(* ---- FB_System_Scenario_Arbitration.st ---- *)
// ==============================================================================
// System scenario arbitration helper
//
// Internal helper for PRG_System.
// Owns scenario request validation, priority resolution, fail-safe clamp,
// degraded-mode adaptation, policy logging, and FB_Scenario_Manager call.
// ==============================================================================
FUNCTION_BLOCK FB_System_Scenario_Arbitration
VAR_INPUT
    VI_System_Time_MS : UDINT;
    VI_IsActivePLC : BOOL;
    VI_System_Mode : E_System_Operating_Mode;
    VI_Security_Armed : BOOL;
END_VAR

VAR_IN_OUT
    VIO_Scenario_Req_Operator : E_SCENARIO_TYPE;
    VIO_Scenario_Req_Gateway : E_SCENARIO_TYPE;
    VIO_Scenario_Req_Rule : E_SCENARIO_TYPE;
    VIO_Scenario_Req_Final : E_SCENARIO_TYPE;
    VIO_Scenario_Intent : E_SCENARIO_TYPE;
    VIO_Scenario_Source : E_SCENARIO_SOURCE;
END_VAR

VAR
    fbLogEvent : FB_LogEvent;
    fbScenarioManager : FB_Scenario_Manager;
END_VAR

// === SCENARIO REQUEST VALIDATION ===
// Normalize invalid values to NONE to avoid corrupt inputs.
// Actual enum range in E_SCENARIO_TYPE is 0..7.
IF TO_USINT(VIO_Scenario_Req_Operator) > 7 THEN
    VIO_Scenario_Req_Operator := E_SCENARIO_TYPE.SCENARIO_NONE;
END_IF;

IF TO_USINT(VIO_Scenario_Req_Gateway) > 7 THEN
    VIO_Scenario_Req_Gateway := E_SCENARIO_TYPE.SCENARIO_NONE;
END_IF;

IF TO_USINT(VIO_Scenario_Req_Rule) > 7 THEN
    VIO_Scenario_Req_Rule := E_SCENARIO_TYPE.SCENARIO_NONE;
END_IF;

// === SCENARIO PRIORITY RESOLUTION ===
// Produces VIO_Scenario_Req_Final (TRACE ONLY, not executed directly)
IF VI_System_Mode = E_System_Operating_Mode.MODE_SAFE_STOP THEN
    VIO_Scenario_Req_Final := 0;
    VIO_Scenario_Source := SRC_SAFETY;
ELSIF VIO_Scenario_Req_Operator <> 0 THEN
    VIO_Scenario_Req_Final := VIO_Scenario_Req_Operator;
    VIO_Scenario_Source := SRC_OPERATOR;
ELSIF VIO_Scenario_Req_Gateway <> 0 THEN
    VIO_Scenario_Req_Final := VIO_Scenario_Req_Gateway;
    VIO_Scenario_Source := SRC_GATEWAY;
ELSIF VIO_Scenario_Req_Rule <> 0 THEN
    VIO_Scenario_Req_Final := VIO_Scenario_Req_Rule;
    VIO_Scenario_Source := SRC_RULE;
ELSE
    VIO_Scenario_Req_Final := GVL_STATUS.G_Current_Scenario;
    VIO_Scenario_Source := SRC_NONE;
END_IF;

VIO_Scenario_Intent := VIO_Scenario_Req_Final;

// === FAIL-SAFE SCENARIO CLAMP ===
CASE VI_System_Mode OF
    E_System_Operating_Mode.MODE_SAFE_STOP:
        VIO_Scenario_Intent := E_SCENARIO_TYPE.SCENARIO_NONE;

    E_System_Operating_Mode.MODE_FREEZE_PROTECTION:
        VIO_Scenario_Intent := E_SCENARIO_TYPE.SCENARIO_NONE;

    E_System_Operating_Mode.MODE_DEGRADED:
        CASE VIO_Scenario_Intent OF
            E_SCENARIO_TYPE.SCENARIO_NONE,
            E_SCENARIO_TYPE.SCENARIO_PRESENCE,
            E_SCENARIO_TYPE.SCENARIO_AWAY,
            E_SCENARIO_TYPE.SCENARIO_SLEEP:
                ; // allowed in degraded
        ELSE
            VIO_Scenario_Intent := E_SCENARIO_TYPE.SCENARIO_NONE;
        END_CASE;
END_CASE;

// === CONTEXT FAIL-SAFE AUTOMATION ===
// If security is armed and no explicit source is requesting another scenario,
// force safe occupancy context to AWAY while system remains in MODE_NORMAL.
IF VI_System_Mode = E_System_Operating_Mode.MODE_NORMAL THEN
    IF VI_Security_Armed AND
       (VIO_Scenario_Req_Operator = E_SCENARIO_TYPE.SCENARIO_NONE) AND
       (VIO_Scenario_Req_Gateway = E_SCENARIO_TYPE.SCENARIO_NONE) AND
       (VIO_Scenario_Req_Rule = E_SCENARIO_TYPE.SCENARIO_NONE) AND
       (VIO_Scenario_Intent <> E_SCENARIO_TYPE.SCENARIO_AWAY) THEN

        IF VIO_Scenario_Intent <> E_SCENARIO_TYPE.SCENARIO_AWAY THEN
            VIO_Scenario_Intent := E_SCENARIO_TYPE.SCENARIO_AWAY;
            VIO_Scenario_Source := SRC_POLICY;

            fbLogEvent(
                VI_Event_Type := 5,
                VI_Timestamp := VI_System_Time_MS,
                VI_Param1 := TO_UDINT(VIO_Scenario_Source),
                VI_Param2 := TO_UDINT(E_SCENARIO_TYPE.SCENARIO_AWAY)
            );
        END_IF;
    END_IF;
END_IF;

// === DEGRADED-AWARE SCENARIO ADAPTATION ===
// Soft adaptation in degraded mode: keep explicit requests intact,
// but if no source is requesting a scenario, move behavior to a safer baseline.
IF VI_System_Mode = E_System_Operating_Mode.MODE_DEGRADED THEN
    IF (VIO_Scenario_Req_Operator = E_SCENARIO_TYPE.SCENARIO_NONE) AND
       (VIO_Scenario_Req_Gateway = E_SCENARIO_TYPE.SCENARIO_NONE) AND
       (VIO_Scenario_Req_Rule = E_SCENARIO_TYPE.SCENARIO_NONE) THEN

        IF VI_Security_Armed THEN
            IF VIO_Scenario_Intent <> E_SCENARIO_TYPE.SCENARIO_AWAY THEN
                VIO_Scenario_Intent := E_SCENARIO_TYPE.SCENARIO_AWAY;
                VIO_Scenario_Source := SRC_POLICY;

                fbLogEvent(
                    VI_Event_Type := 6,
                    VI_Timestamp := VI_System_Time_MS,
                    VI_Param1 := TO_UDINT(VIO_Scenario_Source),
                    VI_Param2 := TO_UDINT(E_SCENARIO_TYPE.SCENARIO_AWAY)
                );
            END_IF;

        ELSIF VIO_Scenario_Intent = E_SCENARIO_TYPE.SCENARIO_PRESENCE THEN
            IF VIO_Scenario_Intent <> E_SCENARIO_TYPE.SCENARIO_SLEEP THEN
                VIO_Scenario_Intent := E_SCENARIO_TYPE.SCENARIO_SLEEP;
                VIO_Scenario_Source := SRC_POLICY;

                fbLogEvent(
                    VI_Event_Type := 7,
                    VI_Timestamp := VI_System_Time_MS,
                    VI_Param1 := TO_UDINT(VIO_Scenario_Source),
                    VI_Param2 := TO_UDINT(E_SCENARIO_TYPE.SCENARIO_SLEEP)
                );
            END_IF;
        END_IF;
    END_IF;
END_IF;

fbScenarioManager(
    VI_System_Time_MS := VI_System_Time_MS,
    VI_Activate_Request := VIO_Scenario_Intent,
    VI_IsActivePLC := VI_IsActivePLC,
    VI_System_Mode := VI_System_Mode,
    VO_Current_Scenario => GVL_STATUS.G_Current_Scenario
);

// >>> BULK_SYNC_ANCHOR: FB_System_Scenario_Arbitration <<<
END_FUNCTION_BLOCK

(* ---- FB_Vent_Output_Projection.st ---- *)
FUNCTION_BLOCK FB_Vent_Output_Projection
VAR_INPUT
    VI_Supply_Fans : ARRAY[1..GVL_CONSTANTS.C_MAX_SUPPLY_FANS] OF BYTE;
    VI_Exhaust_Fans : ARRAY[1..GVL_CONSTANTS.C_MAX_EXHAUST_FANS] OF BYTE;
END_VAR
VAR
    L_i : INT;
END_VAR

// Convert ventilation manager BYTE outputs directly into IO-ready projection.
// PRG_Ventilation no longer needs to publish fan actuator values through GVL_STATE.

FOR L_i := 1 TO GVL_CONSTANTS.C_MAX_SUPPLY_FANS DO
    GVL_VENT_OUTPUT.AO_Supply_Fans[L_i] := BYTE_TO_UINT(VI_Supply_Fans[L_i]) * 10;
END_FOR;

FOR L_i := 1 TO GVL_CONSTANTS.C_MAX_EXHAUST_FANS DO
    GVL_VENT_OUTPUT.AO_Exhaust_Fans[L_i] := BYTE_TO_UINT(VI_Exhaust_Fans[L_i]) * 10;
END_FOR;

END_FUNCTION_BLOCK
// >>> BULK_SYNC_ANCHOR: FB_Vent_Output_Projection <<<

(* ---- MAIN.st ---- *)
PROGRAM MAIN

// ======================================================
// MAIN CYCLIC EXECUTION PIPELINE
// ======================================================
// Required CODESYS Task Configuration:
//   - Assign only PROGRAM MAIN to the cyclic task.
//   - Do not assign child PRG_* programs directly to the same task.
//   - Configure the real cycle time in CODESYS Task Configuration.
//   - Recommended main control cycle: 100 ms.
//
// Execution principle:
//   1. Time / init / configuration
//   2. PLC role arbitration
//   3. IO read and input normalization
//   4. Mode, presence and safety
//   5. Intent, behavior, scenario and policy
//   6. Command arbitration
//   7. Domain execution
//   8. Physical IO write
//   9. Verification, diagnostics, history, HMI
// ======================================================

// 1. Time / init / configuration
PRG_Time_Service();
PRG_System_Init();
PRG_Config_Manager();
PRG_Config_Validation();
PRG_Config_Versioning();
PRG_System_Runtime_Base();

// 2. PLC role arbitration
PRG_PLC_Arbitration();

// 3. IO read and normalized inputs
PRG_IO_Read();
PRG_Input_Processing();

// 4. Base mode, presence and safety
PRG_Mode_Manager();
PRG_Presence_Manager();
PRG_Safety();
PRG_Safety_Operator();
PRG_Safety_Shutdown();
PRG_Safety_Recovery();

// 5. Intent, adaptive behavior, scenario and policy
PRG_System_Intent();
PRG_Security();
PRG_System_Access_Maintenance();
PRG_User_Adapt_Control();
PRG_Behavior_Adapt_Profile();
PRG_Scenario_Engine();
PRG_System_Scenario_Rules();
PRG_System_Evacuation();
PRG_Policy();
PRG_Heating_Policy_Manager();
PRG_Heating_Policy_Observer();
PRG_System_Coordinator();

// 6. Command arbitration
PRG_Command_Arbitration();

// 7. Domain execution and domain output projection
PRG_Heating();
PRG_Ventilation();
PRG_Water();
PRG_Access();
PRG_Lighting();

// 8. Final physical IO projection. Must remain after all domain execution.
PRG_IO_Write();

// 9. Verification, explainability, diagnostics, history, HMI
PRG_Command_Verifier();
PRG_Explainability();
PRG_System_Health();
PRG_System_Alarm_Gateway();
PRG_System_Diagnostics();
PRG_System_Diagnostics_Ext();
PRG_System_History();
PRG_System_BlackBox();
PRG_System_Trend();
PRG_System_Simulation();
PRG_HMI_Dashboard();
PRG_Debug_View();

// >>> BULK_SYNC_ANCHOR: MAIN <<<
END_PROGRAM

(* ---- PRG_Config_Manager.st ---- *)
PROGRAM PRG_Config_Manager
VAR
    L_Error : BOOL;
    L_Index : INT;
END_VAR

L_Error := FALSE;
GVL_CONFIG_VALIDATION.G_Config_Auto_Corrected := FALSE;
GVL_CONFIG_CONTROL.G_Apply_Done := FALSE;
GVL_CONFIG_CONTROL.G_Rollback_Done := FALSE;

IF NOT GVL_CONFIG_SIMULATION.G_Simulation_Result_OK THEN
    GVL_CONFIG_CONTROL.G_Apply_Request := FALSE;
END_IF;

// ===== SIZE VALIDATION =====
IF GVL_SYSTEM_SIZE_CONFIG.G_Active_Heating_Circuits < 1 OR GVL_SYSTEM_SIZE_CONFIG.G_Active_Heating_Circuits > GVL_CONSTANTS.C_MAX_HEATING_CIRCUITS THEN
    GVL_SYSTEM_SIZE_CONFIG.G_Active_Heating_Circuits := GVL_CONSTANTS.C_MAX_HEATING_CIRCUITS;
    L_Error := TRUE;
END_IF;

IF GVL_SYSTEM_SIZE_CONFIG.G_Active_Water_Zones < 1 OR GVL_SYSTEM_SIZE_CONFIG.G_Active_Water_Zones > GVL_CONSTANTS.C_MAX_WATER_ZONES THEN
    GVL_SYSTEM_SIZE_CONFIG.G_Active_Water_Zones := GVL_CONSTANTS.C_MAX_WATER_ZONES;
    L_Error := TRUE;
END_IF;

IF GVL_SYSTEM_SIZE_CONFIG.G_Active_Light_Zones < 1 OR GVL_SYSTEM_SIZE_CONFIG.G_Active_Light_Zones > GVL_CONSTANTS.C_MAX_LIGHT_ZONES THEN
    GVL_SYSTEM_SIZE_CONFIG.G_Active_Light_Zones := GVL_CONSTANTS.C_MAX_LIGHT_ZONES;
    L_Error := TRUE;
END_IF;

// ===== EXISTING VALIDATION =====
IF GVL_INPUT_VALIDATION_CONFIG.G_Reputation_Learning_Rate < 0.0 OR GVL_INPUT_VALIDATION_CONFIG.G_Reputation_Learning_Rate > 1.0 THEN
    GVL_INPUT_VALIDATION_CONFIG.G_Reputation_Learning_Rate := 0.05;
    L_Error := TRUE;
END_IF;

// ===== APPLY (unchanged) =====
IF GVL_CONFIG_CONTROL.G_Apply_Request AND GVL_CONFIG_CONTROL.G_Apply_Confirm THEN
    GVL_CONFIG_CONTROL.BCK_Reputation_Learning_Rate := GVL_INPUT_VALIDATION_CONFIG.G_Reputation_Learning_Rate;
    GVL_INPUT_VALIDATION_CONFIG.G_Reputation_Learning_Rate := GVL_CONFIG_CONTROL.STG_Reputation_Learning_Rate;

    GVL_CONFIG_CONTROL.G_Config_Version := GVL_CONFIG_CONTROL.G_Config_Version + 1;

    L_Index := GVL_CONFIG_HISTORY.G_History_Index;
    GVL_CONFIG_HISTORY.G_History_Version[L_Index] := GVL_CONFIG_CONTROL.G_Config_Version;
    GVL_CONFIG_HISTORY.G_History_Time_MS[L_Index] := GVL_TIME_SERVICE.G_Now_MS;
    GVL_CONFIG_HISTORY.G_History_Action[L_Index] := 'APPLY';

    L_Index := L_Index + 1;
    IF L_Index > 5 THEN L_Index := 1; END_IF;
    GVL_CONFIG_HISTORY.G_History_Index := L_Index;

    GVL_CONFIG_CONTROL.G_Backup_Valid := TRUE;
    GVL_CONFIG_CONTROL.G_Apply_Done := TRUE;
END_IF;

GVL_CONFIG_VALIDATION.G_Config_Valid := NOT L_Error;
GVL_CONFIG_VALIDATION.G_Config_Last_Update_MS := GVL_TIME_SERVICE.G_Now_MS;

// >>> BULK_SYNC_ANCHOR: PRG_Config_Manager <<<
END_PROGRAM

(* ---- PRG_Explainability.st ---- *)
PROGRAM PRG_Explainability
VAR
    L_Mode : E_Safety_Mode;
    L_Recovery : E_Recovery_Phase;
    L_Command : STRING(120);
END_VAR

L_Mode := GVL_SAFETY_SHUTDOWN.G_Safety_Mode;
L_Recovery := GVL_SAFETY_RECOVERY.G_Recovery_Phase;

GVL_EXPLAINABILITY.G_Last_Safety_Mode := L_Mode;
GVL_EXPLAINABILITY.G_Last_Recovery_Phase := L_Recovery;
GVL_EXPLAINABILITY.G_Last_Update_MS := GVL_TIME_SERVICE.G_Now_MS;

// SAFETY LEVEL
CASE L_Mode OF
    FIRE: GVL_EXPLAINABILITY.G_Reason_Chain_Safety := 'FIRE';
    GAS: GVL_EXPLAINABILITY.G_Reason_Chain_Safety := 'GAS';
    WATER_LEAK: GVL_EXPLAINABILITY.G_Reason_Chain_Safety := 'WATER';
    GLOBAL_STOP: GVL_EXPLAINABILITY.G_Reason_Chain_Safety := 'GLOBAL_STOP';
    ELSE
        IF GVL_SAFETY_RECOVERY.G_Recovery_Active THEN
            GVL_EXPLAINABILITY.G_Reason_Chain_Safety := 'RECOVERY';
        ELSE
            GVL_EXPLAINABILITY.G_Reason_Chain_Safety := 'NORMAL';
        END_IF;
END_CASE;

// BEHAVIOR LEVEL
GVL_EXPLAINABILITY.G_Reason_Chain_Behavior := GVL_INTENT_BEHAVIOR.I_Reason_Text;

// COMMAND LEVEL
IF GVL_COMMAND_SHADOW.G_Heating_Block THEN
    L_Command := 'Heating Blocked';
ELSIF GVL_COMMAND_SHADOW.G_Vent_Stop THEN
    L_Command := 'Vent Stopped';
ELSIF GVL_COMMAND_SHADOW.G_Water_Block THEN
    L_Command := 'Water Blocked';
ELSE
    L_Command := 'Command OK';
END_IF;
GVL_EXPLAINABILITY.G_Reason_Chain_Command := L_Command;

// OUTPUT LEVEL
GVL_EXPLAINABILITY.G_Reason_Chain_Output := 'Outputs Applied';

// FULL CHAIN
GVL_EXPLAINABILITY.G_Reason_Chain_Full := CONCAT(CONCAT(CONCAT(GVL_EXPLAINABILITY.G_Reason_Chain_Safety, ' -> '), CONCAT(GVL_EXPLAINABILITY.G_Reason_Chain_Behavior, ' -> ')), CONCAT(GVL_EXPLAINABILITY.G_Reason_Chain_Command, ' -> Outputs Applied'));

// KEEP OLD FIELDS
GVL_EXPLAINABILITY.G_Behavior_Why_Active := GVL_INTENT_BEHAVIOR.I_Reason_Text;

END_PROGRAM

(* ---- PRG_Heating.st ---- *)
PROGRAM PRG_Heating
VAR
    fbHeatingManager : FB_Heating_System_Manager;
    fbDHWManager : FB_DHW_Manager;
    fbOutputProjection : FB_Heating_Output_Projection;

    L_i : INT;
    L_Current_Hour : UINT;
    L_Boiler_Modulation_REAL : ARRAY[1..GVL_CONSTANTS.C_MAX_BOILERS] OF REAL;

    L_Heating_Emergency_Stop : BOOL;
    L_Heating_Gas_Safety_Stop : BOOL;

    L_Zone_Valves : ARRAY[1..GVL_CONSTANTS.C_MAX_HEATING_CIRCUITS] OF BOOL;
    L_Manifold_Pumps : ARRAY[1..GVL_CONSTANTS.C_MAX_MANIFOLDS] OF BOOL;
    L_Manifold_Valves : ARRAY[1..GVL_CONSTANTS.C_MAX_MANIFOLDS] OF REAL;
    L_Boiler_OT_Enable : ARRAY[1..GVL_CONSTANTS.C_MAX_BOILERS] OF BOOL;
    L_Boiler_OT_Setpoint : ARRAY[1..GVL_CONSTANTS.C_MAX_BOILERS] OF REAL;
    L_Backup_Circulation_Pump : BOOL;
    L_Electric_Heater_Enable : BOOL;
    L_Freeze_Risk_Status : BOOL;
    L_Manifold_Status : ARRAY[1..GVL_CONSTANTS.C_MAX_MANIFOLDS] OF ST_Manifold_Status;
    L_Boiler_Status : ARRAY[1..GVL_CONSTANTS.C_MAX_BOILERS] OF ST_Boiler_Status;
    L_DHW_Heating_Pump : BOOL;
    L_DHW_Circ_Pump : BOOL;
    L_DHW_Status : ST_DHW_Status;
END_VAR

// ======================================================
// INPUT ADAPTERS
// ======================================================
FOR L_i := 1 TO GVL_CONSTANTS.C_MAX_BOILERS DO
    L_Boiler_Modulation_REAL[L_i] := TO_REAL(GVL_IO.AI_Boiler_Modulation[L_i]);
END_FOR;

L_Current_Hour := TO_UINT(GVL_TIME_SERVICE.G_Time_Of_Day_MS / 3600000);

L_Heating_Emergency_Stop := GVL_COMMAND_SHADOW.G_Heating_Emergency_Stop;
L_Heating_Gas_Safety_Stop := GVL_COMMAND_SHADOW.G_Heating_Gas_Safety_Stop OR GVL_STATE.G_Safety_Gas_Latched;

// ======================================================
// DHW EXECUTION
// ======================================================
fbDHWManager(
    VI_System_Time_MS := GVL_STATUS.G_System_Time_MS,
    VI_Current_TOD := GVL_STATUS.G_Current_TOD,
    VI_IsActivePLC := GVL_STATUS.G_Is_Active_PLC,
    VI_Temp := GVL_STATE.G_DHW_Temp,
    VI_Pressure := GVL_STATE.G_DHW_Pressure,
    VI_Config := GVL_CONFIG.G_DHW_Config,
    VI_Current_Day_Of_Week := GVL_STATUS.G_Current_Day,
    VI_IO_Modules_Online := GVL_STATUS.G_IO_Modules_Online,
    VI_Reset_Errors := GVL_INTENT_USER.I_Reset_Errors,
    VI_Emergency_Stop := L_Heating_Emergency_Stop,
    VI_System_Mode := GVL_STATE.G_System_Mode,
    VO_Status => L_DHW_Status,
    VO_Heating_Pump => L_DHW_Heating_Pump,
    VO_Circ_Pump => L_DHW_Circ_Pump
);

// Gas safety disables DHW heating demand, but keeps DHW circulation policy intact.
// The electric backup heater is reserved for freeze protection of the heating system, not for DHW.
IF L_Heating_Gas_Safety_Stop THEN
    L_DHW_Heating_Pump := FALSE;
    L_DHW_Status.Heating_Pump_On := FALSE;
END_IF;

// ======================================================
// HEATING EXECUTION CORE
// ======================================================
fbHeatingManager(
    VI_System_Mode := GVL_STATE.G_System_Mode,
    VI_System_Time_MS := GVL_STATUS.G_System_Time_MS,
    VI_IsActivePLC := GVL_STATUS.G_Is_Active_PLC,
    VI_Outdoor_Temp := GVL_STATE.G_Outdoor_Temp,
    VI_Config := GVL_CONFIG.G_Heating_Config,
    VI_Tariff := GVL_CONFIG.G_HMI_Tariff_Settings,
    VI_Current_Hour := L_Current_Hour,
    VI_DHW_Heating_Demand := L_DHW_Heating_Pump,
    VI_DHW_Target_Temp := GVL_CONFIG.G_DHW_Config.Target_Temp,
    VI_Emergency_Stop := L_Heating_Emergency_Stop,
    VI_Gas_Safety_Stop := L_Heating_Gas_Safety_Stop,
    VI_Boiler_Error_Status := GVL_STATE.G_Boiler_Error,
    VI_Boiler_OT_Online := GVL_STATE.G_Boiler_OT_Online,
    VI_Boiler_Modulation := L_Boiler_Modulation_REAL,
    VI_Floor_Temps := GVL_STATE.G_Floor_Temps,
    VI_Room_Temps := GVL_STATE.G_Room_Temps,
    VI_Manifold_Pressures := GVL_STATE.G_Manifold_Pressures,
    VI_Manifold_Currents := GVL_STATE.G_Manifold_Currents,
    VI_Manifold_Temps_Supply := GVL_STATE.G_Manifold_T_Supply,
    VI_Manifold_Temps_Return := GVL_STATE.G_Manifold_T_Return,
    VI_Boiler_Flame_Status := GVL_STATE.G_Boiler_Flame,
    VI_Zone_Configs := GVL_CONFIG.G_HMI_FloorHeating_Configs,
    VI_Rule_Actions := GVL_STATE.G_Rule_Actions,
    VI_IO_Modules_Online := GVL_STATUS.G_IO_Modules_Online,
    VI_Manifold_End_Switches := GVL_STATE.G_Manifold_End_Switches,
    VI_Valve_Test_Config := GVL_CONFIG.G_Valve_Test_Config,
    VO_Manifold_Valves => L_Manifold_Valves,
    VO_Manifold_Pumps => L_Manifold_Pumps,
    VO_Zone_Valves => L_Zone_Valves,
    VO_Boiler_OT_Enable => L_Boiler_OT_Enable,
    VO_Boiler_OT_Setpoint => L_Boiler_OT_Setpoint,
    VO_Backup_Circulation_Pump => L_Backup_Circulation_Pump,
    VO_Electric_Heater_Enable => L_Electric_Heater_Enable,
    VO_Freeze_Risk_Status => L_Freeze_Risk_Status,
    VO_Status => L_Manifold_Status,
    VO_Boiler_Status => L_Boiler_Status
);

// ======================================================
// MAINTENANCE / SERVICE GATING
// ======================================================
GVL_STATUS.G_Diagnostics.Backup_Pump_Out_Of_Service := NOT GVL_CONFIG.G_Backup_Circulation_Pump_In_Service;
GVL_STATUS.G_Diagnostics.Electric_Heater_Out_Of_Service := NOT GVL_CONFIG.G_Electric_Heater_In_Service;

IF NOT GVL_CONFIG.G_Backup_Circulation_Pump_In_Service THEN
    L_Backup_Circulation_Pump := FALSE;
END_IF;

IF NOT GVL_CONFIG.G_Electric_Heater_In_Service THEN
    L_Electric_Heater_Enable := FALSE;
END_IF;

FOR L_i := 1 TO GVL_CONSTANTS.C_MAX_MANIFOLDS DO
    GVL_STATUS.G_Diagnostics.Manifold_Pump_Out_Of_Service[L_i] := NOT GVL_CONFIG.G_Manifold_Pump_In_Service[L_i];
    IF NOT GVL_CONFIG.G_Manifold_Pump_In_Service[L_i] THEN
        L_Manifold_Pumps[L_i] := FALSE;
    END_IF;
END_FOR;

GVL_STATUS.G_Diagnostics.DHW_Heating_Pump_Out_Of_Service := NOT GVL_CONFIG.G_DHW_Heating_Pump_In_Service;
IF NOT GVL_CONFIG.G_DHW_Heating_Pump_In_Service THEN
    L_DHW_Heating_Pump := FALSE;
    L_DHW_Status.Heating_Pump_On := FALSE;
END_IF;

GVL_STATUS.G_Diagnostics.DHW_Circ_Pump_Out_Of_Service := NOT GVL_CONFIG.G_DHW_Circ_Pump_In_Service;
IF NOT GVL_CONFIG.G_DHW_Circ_Pump_In_Service THEN
    L_DHW_Circ_Pump := FALSE;
    L_DHW_Status.Circ_Pump_On := FALSE;
END_IF;

GVL_STATE.G_Freeze_Hardware_Degraded := GVL_STATUS.G_Diagnostics.Backup_Pump_Fault OR GVL_STATUS.G_Diagnostics.Electric_Heater_Fault;
GVL_STATE.G_Freeze_Hardware_Failed := GVL_STATUS.G_Diagnostics.Backup_Pump_Fault AND GVL_STATUS.G_Diagnostics.Electric_Heater_Fault;

IF GVL_STATE.G_Freeze_Hardware_Failed THEN
    L_Backup_Circulation_Pump := FALSE;
    L_Electric_Heater_Enable := FALSE;
    L_Freeze_Risk_Status := TRUE;
END_IF;

// ======================================================
// STATE / STATUS COPY OUT
// ======================================================
FOR L_i := 1 TO GVL_CONSTANTS.C_MAX_HEATING_CIRCUITS DO
    GVL_STATE.G_Zone_Valves[L_i] := L_Zone_Valves[L_i];
END_FOR;

FOR L_i := 1 TO GVL_CONSTANTS.C_MAX_MANIFOLDS DO
    GVL_STATE.G_Manifold_Pumps[L_i] := L_Manifold_Pumps[L_i];
    GVL_STATE.G_Manifold_Valves[L_i] := L_Manifold_Valves[L_i];
    GVL_STATUS.G_Manifold_Status[L_i] := L_Manifold_Status[L_i];
END_FOR;

FOR L_i := 1 TO GVL_CONSTANTS.C_MAX_BOILERS DO
    GVL_STATE.G_Boiler_OT_Enable[L_i] := L_Boiler_OT_Enable[L_i];
    GVL_STATE.G_Boiler_OT_Setpoint[L_i] := L_Boiler_OT_Setpoint[L_i];
    GVL_STATUS.G_Boiler_Status[L_i] := L_Boiler_Status[L_i];
END_FOR;

GVL_STATE.G_Backup_Circulation_Pump := L_Backup_Circulation_Pump;
GVL_STATE.G_Electric_Heater_Enable := L_Electric_Heater_Enable;
GVL_STATE.G_Safety_Freeze_Risk := L_Freeze_Risk_Status;
GVL_STATE.G_DHW_Heating_Pump := L_DHW_Heating_Pump;
GVL_STATE.G_DHW_Circ_Pump := L_DHW_Circ_Pump;
GVL_STATUS.G_DHW_Status := L_DHW_Status;

// ======================================================
// DOMAIN OUTPUT PROJECTION
// ======================================================
fbOutputProjection(
    VI_Zone_Valves := L_Zone_Valves,
    VI_Manifold_Pumps := L_Manifold_Pumps,
    VI_Manifold_Valves := L_Manifold_Valves,
    VI_DHW_Heating_Pump := L_DHW_Heating_Pump,
    VI_DHW_Circ_Pump := L_DHW_Circ_Pump,
    VI_Backup_Circulation_Pump := L_Backup_Circulation_Pump,
    VI_Electric_Heater_Enable := L_Electric_Heater_Enable
);

// >>> BULK_SYNC_ANCHOR: PRG_Heating <<<
END_PROGRAM

(* ---- PRG_HMI_Dashboard.st ---- *)
PROGRAM PRG_HMI_Dashboard
VAR
    L_i : INT;
END_VAR

// Confidence
GVL_HMI.G_HMI_Heating_Confidence := GVL_STATE.G_Heating_Confidence;
GVL_HMI.G_HMI_Heating_Confidence_Percent := REAL_TO_INT(GVL_STATE.G_Heating_Confidence * 100.0);

// Reason
GVL_HMI.G_HMI_Heating_Reason_Code := GVL_STATE.G_Heating_Confidence_Reason_Code;
GVL_HMI.G_HMI_Heating_Status_Text := GVL_STATE.G_Heating_Confidence_Reason_Text;

// Level
IF GVL_STATE.G_Heating_Confidence > 0.8 THEN
    GVL_HMI.G_HMI_Heating_Status_Level := 0;
ELSIF GVL_STATE.G_Heating_Confidence > 0.5 THEN
    GVL_HMI.G_HMI_Heating_Status_Level := 1;
ELSE
    GVL_HMI.G_HMI_Heating_Status_Level := 2;
END_IF;

// Predictive flags
FOR L_i := 1 TO GVL_CONSTANTS.C_MAX_MANIFOLDS DO
    GVL_HMI.G_HMI_Heating_Predictive_Pressure_Drop[L_i] := GVL_STATE.G_Predictive_Pump_Pressure_Drop[L_i];
    GVL_HMI.G_HMI_Heating_Predictive_Current_Rise[L_i] := GVL_STATE.G_Predictive_Pump_Current_Rise[L_i];
END_FOR;

END_PROGRAM
